   STATUS[506].TimeStamp := 16#0000;
   STATUS[507].VALUE := 0.0;
   STATUS[507].TRIGVALUE := 0.0;
   STATUS[507].EXT.AlarmWarnUnAck := FALSE;
   STATUS[507].EXT.AckRequired := FALSE;
   STATUS[507].EXT.Maintanence := FALSE;
   STATUS[507].EXT.Operation := FALSE;
   STATUS[507].EXT.Forced := FALSE;
   STATUS[507].EXT.BIT29 := FALSE;
   STATUS[507].EXT.BIT30 := FALSE;
   STATUS[507].EXT.BIT31 := FALSE;
   STATUS[507].EXT.ModeBit1 := FALSE;
   STATUS[507].EXT.ModeBit2 := FALSE;
   STATUS[507].EXT.ModeBit3 := FALSE;
   STATUS[507].EXT.BIT19 := FALSE;
   STATUS[507].EXT.BIT20 := FALSE;
   STATUS[507].EXT.AlarmSuppressed := FALSE;
   STATUS[507].EXT.AlarmPrsent := FALSE;
   STATUS[507].EXT.AlarmFailUnAck := FALSE;
   STATUS[507].Status := 0;
   STATUS[507].TimeStamp := 16#0000;
   STATUS[508].VALUE := 0.0;
   STATUS[508].TRIGVALUE := 0.0;
   STATUS[508].EXT.AlarmWarnUnAck := FALSE;
   STATUS[508].EXT.AckRequired := FALSE;
   STATUS[508].EXT.Maintanence := FALSE;
   STATUS[508].EXT.Operation := FALSE;
   STATUS[508].EXT.Forced := FALSE;
   STATUS[508].EXT.BIT29 := FALSE;
   STATUS[508].EXT.BIT30 := FALSE;
   STATUS[508].EXT.BIT31 := FALSE;
   STATUS[508].EXT.ModeBit1 := FALSE;
   STATUS[508].EXT.ModeBit2 := FALSE;
   STATUS[508].EXT.ModeBit3 := FALSE;
   STATUS[508].EXT.BIT19 := FALSE;
   STATUS[508].EXT.BIT20 := FALSE;
   STATUS[508].EXT.AlarmSuppressed := FALSE;
   STATUS[508].EXT.AlarmPrsent := FALSE;
   STATUS[508].EXT.AlarmFailUnAck := FALSE;
   STATUS[508].Status := 0;
   STATUS[508].TimeStamp := 16#0000;
   STATUS[509].VALUE := 0.0;
   STATUS[509].TRIGVALUE := 0.0;
   STATUS[509].EXT.AlarmWarnUnAck := FALSE;
   STATUS[509].EXT.AckRequired := FALSE;
   STATUS[509].EXT.Maintanence := FALSE;
   STATUS[509].EXT.Operation := FALSE;
   STATUS[509].EXT.Forced := FALSE;
   STATUS[509].EXT.BIT29 := FALSE;
   STATUS[509].EXT.BIT30 := FALSE;
   STATUS[509].EXT.BIT31 := FALSE;
   STATUS[509].EXT.ModeBit1 := FALSE;
   STATUS[509].EXT.ModeBit2 := FALSE;
   STATUS[509].EXT.ModeBit3 := FALSE;
   STATUS[509].EXT.BIT19 := FALSE;
   STATUS[509].EXT.BIT20 := FALSE;
   STATUS[509].EXT.AlarmSuppressed := FALSE;
   STATUS[509].EXT.AlarmPrsent := FALSE;
   STATUS[509].EXT.AlarmFailUnAck := FALSE;
   STATUS[509].Status := 0;
   STATUS[509].TimeStamp := 16#0000;
   STATUS[510].VALUE := 0.0;
   STATUS[510].TRIGVALUE := 0.0;
   STATUS[510].EXT.AlarmWarnUnAck := FALSE;
   STATUS[510].EXT.AckRequired := FALSE;
   STATUS[510].EXT.Maintanence := FALSE;
   STATUS[510].EXT.Operation := FALSE;
   STATUS[510].EXT.Forced := FALSE;
   STATUS[510].EXT.BIT29 := FALSE;
   STATUS[510].EXT.BIT30 := FALSE;
   STATUS[510].EXT.BIT31 := FALSE;
   STATUS[510].EXT.ModeBit1 := FALSE;
   STATUS[510].EXT.ModeBit2 := FALSE;
   STATUS[510].EXT.ModeBit3 := FALSE;
   STATUS[510].EXT.BIT19 := FALSE;
   STATUS[510].EXT.BIT20 := FALSE;
   STATUS[510].EXT.AlarmSuppressed := FALSE;
   STATUS[510].EXT.AlarmPrsent := FALSE;
   STATUS[510].EXT.AlarmFailUnAck := FALSE;
   STATUS[510].Status := 0;
   STATUS[510].TimeStamp := 16#0000;
   STATUS[511].VALUE := 0.0;
   STATUS[511].TRIGVALUE := 0.0;
   STATUS[511].EXT.AlarmWarnUnAck := FALSE;
   STATUS[511].EXT.AckRequired := FALSE;
   STATUS[511].EXT.Maintanence := FALSE;
   STATUS[511].EXT.Operation := FALSE;
   STATUS[511].EXT.Forced := FALSE;
   STATUS[511].EXT.BIT29 := FALSE;
   STATUS[511].EXT.BIT30 := FALSE;
   STATUS[511].EXT.BIT31 := FALSE;
   STATUS[511].EXT.ModeBit1 := FALSE;
   STATUS[511].EXT.ModeBit2 := FALSE;
   STATUS[511].EXT.ModeBit3 := FALSE;
   STATUS[511].EXT.BIT19 := FALSE;
   STATUS[511].EXT.BIT20 := FALSE;
   STATUS[511].EXT.AlarmSuppressed := FALSE;
   STATUS[511].EXT.AlarmPrsent := FALSE;
   STATUS[511].EXT.AlarmFailUnAck := FALSE;
   STATUS[511].Status := 0;
   STATUS[511].TimeStamp := 16#0000;
   STATUS[512].VALUE := 0.0;
   STATUS[512].TRIGVALUE := 0.0;
   STATUS[512].EXT.AlarmWarnUnAck := FALSE;
   STATUS[512].EXT.AckRequired := FALSE;
   STATUS[512].EXT.Maintanence := FALSE;
   STATUS[512].EXT.Operation := FALSE;
   STATUS[512].EXT.Forced := FALSE;
   STATUS[512].EXT.BIT29 := FALSE;
   STATUS[512].EXT.BIT30 := FALSE;
   STATUS[512].EXT.BIT31 := FALSE;
   STATUS[512].EXT.ModeBit1 := FALSE;
   STATUS[512].EXT.ModeBit2 := FALSE;
   STATUS[512].EXT.ModeBit3 := FALSE;
   STATUS[512].EXT.BIT19 := FALSE;
   STATUS[512].EXT.BIT20 := FALSE;
   STATUS[512].EXT.AlarmSuppressed := FALSE;
   STATUS[512].EXT.AlarmPrsent := FALSE;
   STATUS[512].EXT.AlarmFailUnAck := FALSE;
   STATUS[512].Status := 0;
   STATUS[512].TimeStamp := 16#0000;
   STATUS[513].VALUE := 0.0;
   STATUS[513].TRIGVALUE := 0.0;
   STATUS[513].EXT.AlarmWarnUnAck := FALSE;
   STATUS[513].EXT.AckRequired := FALSE;
   STATUS[513].EXT.Maintanence := FALSE;
   STATUS[513].EXT.Operation := FALSE;
   STATUS[513].EXT.Forced := FALSE;
   STATUS[513].EXT.BIT29 := FALSE;
   STATUS[513].EXT.BIT30 := FALSE;
   STATUS[513].EXT.BIT31 := FALSE;
   STATUS[513].EXT.ModeBit1 := FALSE;
   STATUS[513].EXT.ModeBit2 := FALSE;
   STATUS[513].EXT.ModeBit3 := FALSE;
   STATUS[513].EXT.BIT19 := FALSE;
   STATUS[513].EXT.BIT20 := FALSE;
   STATUS[513].EXT.AlarmSuppressed := FALSE;
   STATUS[513].EXT.AlarmPrsent := FALSE;
   STATUS[513].EXT.AlarmFailUnAck := FALSE;
   STATUS[513].Status := 0;
   STATUS[513].TimeStamp := 16#0000;
   STATUS[514].VALUE := 0.0;
   STATUS[514].TRIGVALUE := 0.0;
   STATUS[514].EXT.AlarmWarnUnAck := FALSE;
   STATUS[514].EXT.AckRequired := FALSE;
   STATUS[514].EXT.Maintanence := FALSE;
   STATUS[514].EXT.Operation := FALSE;
   STATUS[514].EXT.Forced := FALSE;
   STATUS[514].EXT.BIT29 := FALSE;
   STATUS[514].EXT.BIT30 := FALSE;
   STATUS[514].EXT.BIT31 := FALSE;
   STATUS[514].EXT.ModeBit1 := FALSE;
   STATUS[514].EXT.ModeBit2 := FALSE;
   STATUS[514].EXT.ModeBit3 := FALSE;
   STATUS[514].EXT.BIT19 := FALSE;
   STATUS[514].EXT.BIT20 := FALSE;
   STATUS[514].EXT.AlarmSuppressed := FALSE;
   STATUS[514].EXT.AlarmPrsent := FALSE;
   STATUS[514].EXT.AlarmFailUnAck := FALSE;
   STATUS[514].Status := 0;
   STATUS[514].TimeStamp := 16#0000;
   STATUS[515].VALUE := 0.0;
   STATUS[515].TRIGVALUE := 0.0;
   STATUS[515].EXT.AlarmWarnUnAck := FALSE;
   STATUS[515].EXT.AckRequired := FALSE;
   STATUS[515].EXT.Maintanence := FALSE;
   STATUS[515].EXT.Operation := FALSE;
   STATUS[515].EXT.Forced := FALSE;
   STATUS[515].EXT.BIT29 := FALSE;
   STATUS[515].EXT.BIT30 := FALSE;
   STATUS[515].EXT.BIT31 := FALSE;
   STATUS[515].EXT.ModeBit1 := FALSE;
   STATUS[515].EXT.ModeBit2 := FALSE;
   STATUS[515].EXT.ModeBit3 := FALSE;
   STATUS[515].EXT.BIT19 := FALSE;
   STATUS[515].EXT.BIT20 := FALSE;
   STATUS[515].EXT.AlarmSuppressed := FALSE;
   STATUS[515].EXT.AlarmPrsent := FALSE;
   STATUS[515].EXT.AlarmFailUnAck := FALSE;
   STATUS[515].Status := 0;
   STATUS[515].TimeStamp := 16#0000;
   STATUS[516].VALUE := 0.0;
   STATUS[516].TRIGVALUE := 0.0;
   STATUS[516].EXT.AlarmWarnUnAck := FALSE;
   STATUS[516].EXT.AckRequired := FALSE;
   STATUS[516].EXT.Maintanence := FALSE;
   STATUS[516].EXT.Operation := FALSE;
   STATUS[516].EXT.Forced := FALSE;
   STATUS[516].EXT.BIT29 := FALSE;
   STATUS[516].EXT.BIT30 := FALSE;
   STATUS[516].EXT.BIT31 := FALSE;
   STATUS[516].EXT.ModeBit1 := FALSE;
   STATUS[516].EXT.ModeBit2 := FALSE;
   STATUS[516].EXT.ModeBit3 := FALSE;
   STATUS[516].EXT.BIT19 := FALSE;
   STATUS[516].EXT.BIT20 := FALSE;
   STATUS[516].EXT.AlarmSuppressed := FALSE;
   STATUS[516].EXT.AlarmPrsent := FALSE;
   STATUS[516].EXT.AlarmFailUnAck := FALSE;
   STATUS[516].Status := 0;
   STATUS[516].TimeStamp := 16#0000;
   STATUS[517].VALUE := 0.0;
   STATUS[517].TRIGVALUE := 0.0;
   STATUS[517].EXT.AlarmWarnUnAck := FALSE;
   STATUS[517].EXT.AckRequired := FALSE;
   STATUS[517].EXT.Maintanence := FALSE;
   STATUS[517].EXT.Operation := FALSE;
   STATUS[517].EXT.Forced := FALSE;
   STATUS[517].EXT.BIT29 := FALSE;
   STATUS[517].EXT.BIT30 := FALSE;
   STATUS[517].EXT.BIT31 := FALSE;
   STATUS[517].EXT.ModeBit1 := FALSE;
   STATUS[517].EXT.ModeBit2 := FALSE;
   STATUS[517].EXT.ModeBit3 := FALSE;
   STATUS[517].EXT.BIT19 := FALSE;
   STATUS[517].EXT.BIT20 := FALSE;
   STATUS[517].EXT.AlarmSuppressed := FALSE;
   STATUS[517].EXT.AlarmPrsent := FALSE;
   STATUS[517].EXT.AlarmFailUnAck := FALSE;
   STATUS[517].Status := 0;
   STATUS[517].TimeStamp := 16#0000;
   STATUS[518].VALUE := 0.0;
   STATUS[518].TRIGVALUE := 0.0;
   STATUS[518].EXT.AlarmWarnUnAck := FALSE;
   STATUS[518].EXT.AckRequired := FALSE;
   STATUS[518].EXT.Maintanence := FALSE;
   STATUS[518].EXT.Operation := FALSE;
   STATUS[518].EXT.Forced := FALSE;
   STATUS[518].EXT.BIT29 := FALSE;
   STATUS[518].EXT.BIT30 := FALSE;
   STATUS[518].EXT.BIT31 := FALSE;
   STATUS[518].EXT.ModeBit1 := FALSE;
   STATUS[518].EXT.ModeBit2 := FALSE;
   STATUS[518].EXT.ModeBit3 := FALSE;
   STATUS[518].EXT.BIT19 := FALSE;
   STATUS[518].EXT.BIT20 := FALSE;
   STATUS[518].EXT.AlarmSuppressed := FALSE;
   STATUS[518].EXT.AlarmPrsent := FALSE;
   STATUS[518].EXT.AlarmFailUnAck := FALSE;
   STATUS[518].Status := 0;
   STATUS[518].TimeStamp := 16#0000;
   STATUS[519].VALUE := 0.0;
   STATUS[519].TRIGVALUE := 0.0;
   STATUS[519].EXT.AlarmWarnUnAck := FALSE;
   STATUS[519].EXT.AckRequired := FALSE;
   STATUS[519].EXT.Maintanence := FALSE;
   STATUS[519].EXT.Operation := FALSE;
   STATUS[519].EXT.Forced := FALSE;
   STATUS[519].EXT.BIT29 := FALSE;
   STATUS[519].EXT.BIT30 := FALSE;
   STATUS[519].EXT.BIT31 := FALSE;
   STATUS[519].EXT.ModeBit1 := FALSE;
   STATUS[519].EXT.ModeBit2 := FALSE;
   STATUS[519].EXT.ModeBit3 := FALSE;
   STATUS[519].EXT.BIT19 := FALSE;
   STATUS[519].EXT.BIT20 := FALSE;
   STATUS[519].EXT.AlarmSuppressed := FALSE;
   STATUS[519].EXT.AlarmPrsent := FALSE;
   STATUS[519].EXT.AlarmFailUnAck := FALSE;
   STATUS[519].Status := 0;
   STATUS[519].TimeStamp := 16#0000;
   STATUS[520].VALUE := 0.0;
   STATUS[520].TRIGVALUE := 0.0;
   STATUS[520].EXT.AlarmWarnUnAck := FALSE;
   STATUS[520].EXT.AckRequired := FALSE;
   STATUS[520].EXT.Maintanence := FALSE;
   STATUS[520].EXT.Operation := FALSE;
   STATUS[520].EXT.Forced := FALSE;
   STATUS[520].EXT.BIT29 := FALSE;
   STATUS[520].EXT.BIT30 := FALSE;
   STATUS[520].EXT.BIT31 := FALSE;
   STATUS[520].EXT.ModeBit1 := FALSE;
   STATUS[520].EXT.ModeBit2 := FALSE;
   STATUS[520].EXT.ModeBit3 := FALSE;
   STATUS[520].EXT.BIT19 := FALSE;
   STATUS[520].EXT.BIT20 := FALSE;
   STATUS[520].EXT.AlarmSuppressed := FALSE;
   STATUS[520].EXT.AlarmPrsent := FALSE;
   STATUS[520].EXT.AlarmFailUnAck := FALSE;
   STATUS[520].Status := 0;
   STATUS[520].TimeStamp := 16#0000;
   STATUS[521].VALUE := 0.0;
   STATUS[521].TRIGVALUE := 0.0;
   STATUS[521].EXT.AlarmWarnUnAck := FALSE;
   STATUS[521].EXT.AckRequired := FALSE;
   STATUS[521].EXT.Maintanence := FALSE;
   STATUS[521].EXT.Operation := FALSE;
   STATUS[521].EXT.Forced := FALSE;
   STATUS[521].EXT.BIT29 := FALSE;
   STATUS[521].EXT.BIT30 := FALSE;
   STATUS[521].EXT.BIT31 := FALSE;
   STATUS[521].EXT.ModeBit1 := FALSE;
   STATUS[521].EXT.ModeBit2 := FALSE;
   STATUS[521].EXT.ModeBit3 := FALSE;
   STATUS[521].EXT.BIT19 := FALSE;
   STATUS[521].EXT.BIT20 := FALSE;
   STATUS[521].EXT.AlarmSuppressed := FALSE;
   STATUS[521].EXT.AlarmPrsent := FALSE;
   STATUS[521].EXT.AlarmFailUnAck := FALSE;
   STATUS[521].Status := 0;
   STATUS[521].TimeStamp := 16#0000;
   STATUS[522].VALUE := 0.0;
   STATUS[522].TRIGVALUE := 0.0;
   STATUS[522].EXT.AlarmWarnUnAck := FALSE;
   STATUS[522].EXT.AckRequired := FALSE;
   STATUS[522].EXT.Maintanence := FALSE;
   STATUS[522].EXT.Operation := FALSE;
   STATUS[522].EXT.Forced := FALSE;
   STATUS[522].EXT.BIT29 := FALSE;
   STATUS[522].EXT.BIT30 := FALSE;
   STATUS[522].EXT.BIT31 := FALSE;
   STATUS[522].EXT.ModeBit1 := FALSE;
   STATUS[522].EXT.ModeBit2 := FALSE;
   STATUS[522].EXT.ModeBit3 := FALSE;
   STATUS[522].EXT.BIT19 := FALSE;
   STATUS[522].EXT.BIT20 := FALSE;
   STATUS[522].EXT.AlarmSuppressed := FALSE;
   STATUS[522].EXT.AlarmPrsent := FALSE;
   STATUS[522].EXT.AlarmFailUnAck := FALSE;
   STATUS[522].Status := 0;
   STATUS[522].TimeStamp := 16#0000;
   STATUS[523].VALUE := 0.0;
   STATUS[523].TRIGVALUE := 0.0;
   STATUS[523].EXT.AlarmWarnUnAck := FALSE;
   STATUS[523].EXT.AckRequired := FALSE;
   STATUS[523].EXT.Maintanence := FALSE;
   STATUS[523].EXT.Operation := FALSE;
   STATUS[523].EXT.Forced := FALSE;
   STATUS[523].EXT.BIT29 := FALSE;
   STATUS[523].EXT.BIT30 := FALSE;
   STATUS[523].EXT.BIT31 := FALSE;
   STATUS[523].EXT.ModeBit1 := FALSE;
   STATUS[523].EXT.ModeBit2 := FALSE;
   STATUS[523].EXT.ModeBit3 := FALSE;
   STATUS[523].EXT.BIT19 := FALSE;
   STATUS[523].EXT.BIT20 := FALSE;
   STATUS[523].EXT.AlarmSuppressed := FALSE;
   STATUS[523].EXT.AlarmPrsent := FALSE;
   STATUS[523].EXT.AlarmFailUnAck := FALSE;
   STATUS[523].Status := 0;
   STATUS[523].TimeStamp := 16#0000;
   STATUS[524].VALUE := 0.0;
   STATUS[524].TRIGVALUE := 0.0;
   STATUS[524].EXT.AlarmWarnUnAck := FALSE;
   STATUS[524].EXT.AckRequired := FALSE;
   STATUS[524].EXT.Maintanence := FALSE;
   STATUS[524].EXT.Operation := FALSE;
   STATUS[524].EXT.Forced := FALSE;
   STATUS[524].EXT.BIT29 := FALSE;
   STATUS[524].EXT.BIT30 := FALSE;
   STATUS[524].EXT.BIT31 := FALSE;
   STATUS[524].EXT.ModeBit1 := FALSE;
   STATUS[524].EXT.ModeBit2 := FALSE;
   STATUS[524].EXT.ModeBit3 := FALSE;
   STATUS[524].EXT.BIT19 := FALSE;
   STATUS[524].EXT.BIT20 := FALSE;
   STATUS[524].EXT.AlarmSuppressed := FALSE;
   STATUS[524].EXT.AlarmPrsent := FALSE;
   STATUS[524].EXT.AlarmFailUnAck := FALSE;
   STATUS[524].Status := 0;
   STATUS[524].TimeStamp := 16#0000;
   STATUS[525].VALUE := 0.0;
   STATUS[525].TRIGVALUE := 0.0;
   STATUS[525].EXT.AlarmWarnUnAck := FALSE;
   STATUS[525].EXT.AckRequired := FALSE;
   STATUS[525].EXT.Maintanence := FALSE;
   STATUS[525].EXT.Operation := FALSE;
   STATUS[525].EXT.Forced := FALSE;
   STATUS[525].EXT.BIT29 := FALSE;
   STATUS[525].EXT.BIT30 := FALSE;
   STATUS[525].EXT.BIT31 := FALSE;
   STATUS[525].EXT.ModeBit1 := FALSE;
   STATUS[525].EXT.ModeBit2 := FALSE;
   STATUS[525].EXT.ModeBit3 := FALSE;
   STATUS[525].EXT.BIT19 := FALSE;
   STATUS[525].EXT.BIT20 := FALSE;
   STATUS[525].EXT.AlarmSuppressed := FALSE;
   STATUS[525].EXT.AlarmPrsent := FALSE;
   STATUS[525].EXT.AlarmFailUnAck := FALSE;
   STATUS[525].Status := 0;
   STATUS[525].TimeStamp := 16#0000;
   STATUS[526].VALUE := 0.0;
   STATUS[526].TRIGVALUE := 0.0;
   STATUS[526].EXT.AlarmWarnUnAck := FALSE;
   STATUS[526].EXT.AckRequired := FALSE;
   STATUS[526].EXT.Maintanence := FALSE;
   STATUS[526].EXT.Operation := FALSE;
   STATUS[526].EXT.Forced := FALSE;
   STATUS[526].EXT.BIT29 := FALSE;
   STATUS[526].EXT.BIT30 := FALSE;
   STATUS[526].EXT.BIT31 := FALSE;
   STATUS[526].EXT.ModeBit1 := FALSE;
   STATUS[526].EXT.ModeBit2 := FALSE;
   STATUS[526].EXT.ModeBit3 := FALSE;
   STATUS[526].EXT.BIT19 := FALSE;
   STATUS[526].EXT.BIT20 := FALSE;
   STATUS[526].EXT.AlarmSuppressed := FALSE;
   STATUS[526].EXT.AlarmPrsent := FALSE;
   STATUS[526].EXT.AlarmFailUnAck := FALSE;
   STATUS[526].Status := 0;
   STATUS[526].TimeStamp := 16#0000;
   STATUS[527].VALUE := 0.0;
   STATUS[527].TRIGVALUE := 0.0;
   STATUS[527].EXT.AlarmWarnUnAck := FALSE;
   STATUS[527].EXT.AckRequired := FALSE;
   STATUS[527].EXT.Maintanence := FALSE;
   STATUS[527].EXT.Operation := FALSE;
   STATUS[527].EXT.Forced := FALSE;
   STATUS[527].EXT.BIT29 := FALSE;
   STATUS[527].EXT.BIT30 := FALSE;
   STATUS[527].EXT.BIT31 := FALSE;
   STATUS[527].EXT.ModeBit1 := FALSE;
   STATUS[527].EXT.ModeBit2 := FALSE;
   STATUS[527].EXT.ModeBit3 := FALSE;
   STATUS[527].EXT.BIT19 := FALSE;
   STATUS[527].EXT.BIT20 := FALSE;
   STATUS[527].EXT.AlarmSuppressed := FALSE;
   STATUS[527].EXT.AlarmPrsent := FALSE;
   STATUS[527].EXT.AlarmFailUnAck := FALSE;
   STATUS[527].Status := 0;
   STATUS[527].TimeStamp := 16#0000;
   STATUS[528].VALUE := 0.0;
   STATUS[528].TRIGVALUE := 0.0;
   STATUS[528].EXT.AlarmWarnUnAck := FALSE;
   STATUS[528].EXT.AckRequired := FALSE;
   STATUS[528].EXT.Maintanence := FALSE;
   STATUS[528].EXT.Operation := FALSE;
   STATUS[528].EXT.Forced := FALSE;
   STATUS[528].EXT.BIT29 := FALSE;
   STATUS[528].EXT.BIT30 := FALSE;
   STATUS[528].EXT.BIT31 := FALSE;
   STATUS[528].EXT.ModeBit1 := FALSE;
   STATUS[528].EXT.ModeBit2 := FALSE;
   STATUS[528].EXT.ModeBit3 := FALSE;
   STATUS[528].EXT.BIT19 := FALSE;
   STATUS[528].EXT.BIT20 := FALSE;
   STATUS[528].EXT.AlarmSuppressed := FALSE;
   STATUS[528].EXT.AlarmPrsent := FALSE;
   STATUS[528].EXT.AlarmFailUnAck := FALSE;
   STATUS[528].Status := 0;
   STATUS[528].TimeStamp := 16#0000;
   STATUS[529].VALUE := 0.0;
   STATUS[529].TRIGVALUE := 0.0;
   STATUS[529].EXT.AlarmWarnUnAck := FALSE;
   STATUS[529].EXT.AckRequired := FALSE;
   STATUS[529].EXT.Maintanence := FALSE;
   STATUS[529].EXT.Operation := FALSE;
   STATUS[529].EXT.Forced := FALSE;
   STATUS[529].EXT.BIT29 := FALSE;
   STATUS[529].EXT.BIT30 := FALSE;
   STATUS[529].EXT.BIT31 := FALSE;
   STATUS[529].EXT.ModeBit1 := FALSE;
   STATUS[529].EXT.ModeBit2 := FALSE;
   STATUS[529].EXT.ModeBit3 := FALSE;
   STATUS[529].EXT.BIT19 := FALSE;
   STATUS[529].EXT.BIT20 := FALSE;
   STATUS[529].EXT.AlarmSuppressed := FALSE;
   STATUS[529].EXT.AlarmPrsent := FALSE;
   STATUS[529].EXT.AlarmFailUnAck := FALSE;
   STATUS[529].Status := 0;
   STATUS[529].TimeStamp := 16#0000;
   STATUS[530].VALUE := 0.0;
   STATUS[530].TRIGVALUE := 0.0;
   STATUS[530].EXT.AlarmWarnUnAck := FALSE;
   STATUS[530].EXT.AckRequired := FALSE;
   STATUS[530].EXT.Maintanence := FALSE;
   STATUS[530].EXT.Operation := FALSE;
   STATUS[530].EXT.Forced := FALSE;
   STATUS[530].EXT.BIT29 := FALSE;
   STATUS[530].EXT.BIT30 := FALSE;
   STATUS[530].EXT.BIT31 := FALSE;
   STATUS[530].EXT.ModeBit1 := FALSE;
   STATUS[530].EXT.ModeBit2 := FALSE;
   STATUS[530].EXT.ModeBit3 := FALSE;
   STATUS[530].EXT.BIT19 := FALSE;
   STATUS[530].EXT.BIT20 := FALSE;
   STATUS[530].EXT.AlarmSuppressed := FALSE;
   STATUS[530].EXT.AlarmPrsent := FALSE;
   STATUS[530].EXT.AlarmFailUnAck := FALSE;
   STATUS[530].Status := 0;
   STATUS[530].TimeStamp := 16#0000;
   STATUS[531].VALUE := 0.0;
   STATUS[531].TRIGVALUE := 0.0;
   STATUS[531].EXT.AlarmWarnUnAck := FALSE;
   STATUS[531].EXT.AckRequired := FALSE;
   STATUS[531].EXT.Maintanence := FALSE;
   STATUS[531].EXT.Operation := FALSE;
   STATUS[531].EXT.Forced := FALSE;
   STATUS[531].EXT.BIT29 := FALSE;
   STATUS[531].EXT.BIT30 := FALSE;
   STATUS[531].EXT.BIT31 := FALSE;
   STATUS[531].EXT.ModeBit1 := FALSE;
   STATUS[531].EXT.ModeBit2 := FALSE;
   STATUS[531].EXT.ModeBit3 := FALSE;
   STATUS[531].EXT.BIT19 := FALSE;
   STATUS[531].EXT.BIT20 := FALSE;
   STATUS[531].EXT.AlarmSuppressed := FALSE;
   STATUS[531].EXT.AlarmPrsent := FALSE;
   STATUS[531].EXT.AlarmFailUnAck := FALSE;
   STATUS[531].Status := 0;
   STATUS[531].TimeStamp := 16#0000;
   STATUS[532].VALUE := 0.0;
   STATUS[532].TRIGVALUE := 0.0;
   STATUS[532].EXT.AlarmWarnUnAck := FALSE;
   STATUS[532].EXT.AckRequired := FALSE;
   STATUS[532].EXT.Maintanence := FALSE;
   STATUS[532].EXT.Operation := FALSE;
   STATUS[532].EXT.Forced := FALSE;
   STATUS[532].EXT.BIT29 := FALSE;
   STATUS[532].EXT.BIT30 := FALSE;
   STATUS[532].EXT.BIT31 := FALSE;
   STATUS[532].EXT.ModeBit1 := FALSE;
   STATUS[532].EXT.ModeBit2 := FALSE;
   STATUS[532].EXT.ModeBit3 := FALSE;
   STATUS[532].EXT.BIT19 := FALSE;
   STATUS[532].EXT.BIT20 := FALSE;
   STATUS[532].EXT.AlarmSuppressed := FALSE;
   STATUS[532].EXT.AlarmPrsent := FALSE;
   STATUS[532].EXT.AlarmFailUnAck := FALSE;
   STATUS[532].Status := 0;
   STATUS[532].TimeStamp := 16#0000;
   STATUS[533].VALUE := 0.0;
   STATUS[533].TRIGVALUE := 0.0;
   STATUS[533].EXT.AlarmWarnUnAck := FALSE;
   STATUS[533].EXT.AckRequired := FALSE;
   STATUS[533].EXT.Maintanence := FALSE;
   STATUS[533].EXT.Operation := FALSE;
   STATUS[533].EXT.Forced := FALSE;
   STATUS[533].EXT.BIT29 := FALSE;
   STATUS[533].EXT.BIT30 := FALSE;
   STATUS[533].EXT.BIT31 := FALSE;
   STATUS[533].EXT.ModeBit1 := FALSE;
   STATUS[533].EXT.ModeBit2 := FALSE;
   STATUS[533].EXT.ModeBit3 := FALSE;
   STATUS[533].EXT.BIT19 := FALSE;
   STATUS[533].EXT.BIT20 := FALSE;
   STATUS[533].EXT.AlarmSuppressed := FALSE;
   STATUS[533].EXT.AlarmPrsent := FALSE;
   STATUS[533].EXT.AlarmFailUnAck := FALSE;
   STATUS[533].Status := 0;
   STATUS[533].TimeStamp := 16#0000;
   STATUS[534].VALUE := 0.0;
   STATUS[534].TRIGVALUE := 0.0;
   STATUS[534].EXT.AlarmWarnUnAck := FALSE;
   STATUS[534].EXT.AckRequired := FALSE;
   STATUS[534].EXT.Maintanence := FALSE;
   STATUS[534].EXT.Operation := FALSE;
   STATUS[534].EXT.Forced := FALSE;
   STATUS[534].EXT.BIT29 := FALSE;
   STATUS[534].EXT.BIT30 := FALSE;
   STATUS[534].EXT.BIT31 := FALSE;
   STATUS[534].EXT.ModeBit1 := FALSE;
   STATUS[534].EXT.ModeBit2 := FALSE;
   STATUS[534].EXT.ModeBit3 := FALSE;
   STATUS[534].EXT.BIT19 := FALSE;
   STATUS[534].EXT.BIT20 := FALSE;
   STATUS[534].EXT.AlarmSuppressed := FALSE;
   STATUS[534].EXT.AlarmPrsent := FALSE;
   STATUS[534].EXT.AlarmFailUnAck := FALSE;
   STATUS[534].Status := 0;
   STATUS[534].TimeStamp := 16#0000;
   STATUS[535].VALUE := 0.0;
   STATUS[535].TRIGVALUE := 0.0;
   STATUS[535].EXT.AlarmWarnUnAck := FALSE;
   STATUS[535].EXT.AckRequired := FALSE;
   STATUS[535].EXT.Maintanence := FALSE;
   STATUS[535].EXT.Operation := FALSE;
   STATUS[535].EXT.Forced := FALSE;
   STATUS[535].EXT.BIT29 := FALSE;
   STATUS[535].EXT.BIT30 := FALSE;
   STATUS[535].EXT.BIT31 := FALSE;
   STATUS[535].EXT.ModeBit1 := FALSE;
   STATUS[535].EXT.ModeBit2 := FALSE;
   STATUS[535].EXT.ModeBit3 := FALSE;
   STATUS[535].EXT.BIT19 := FALSE;
   STATUS[535].EXT.BIT20 := FALSE;
   STATUS[535].EXT.AlarmSuppressed := FALSE;
   STATUS[535].EXT.AlarmPrsent := FALSE;
   STATUS[535].EXT.AlarmFailUnAck := FALSE;
   STATUS[535].Status := 0;
   STATUS[535].TimeStamp := 16#0000;
   STATUS[536].VALUE := 0.0;
   STATUS[536].TRIGVALUE := 0.0;
   STATUS[536].EXT.AlarmWarnUnAck := FALSE;
   STATUS[536].EXT.AckRequired := FALSE;
   STATUS[536].EXT.Maintanence := FALSE;
   STATUS[536].EXT.Operation := FALSE;
   STATUS[536].EXT.Forced := FALSE;
   STATUS[536].EXT.BIT29 := FALSE;
   STATUS[536].EXT.BIT30 := FALSE;
   STATUS[536].EXT.BIT31 := FALSE;
   STATUS[536].EXT.ModeBit1 := FALSE;
   STATUS[536].EXT.ModeBit2 := FALSE;
   STATUS[536].EXT.ModeBit3 := FALSE;
   STATUS[536].EXT.BIT19 := FALSE;
   STATUS[536].EXT.BIT20 := FALSE;
   STATUS[536].EXT.AlarmSuppressed := FALSE;
   STATUS[536].EXT.AlarmPrsent := FALSE;
   STATUS[536].EXT.AlarmFailUnAck := FALSE;
   STATUS[536].Status := 0;
   STATUS[536].TimeStamp := 16#0000;
   STATUS[537].VALUE := 0.0;
   STATUS[537].TRIGVALUE := 0.0;
   STATUS[537].EXT.AlarmWarnUnAck := FALSE;
   STATUS[537].EXT.AckRequired := FALSE;
   STATUS[537].EXT.Maintanence := FALSE;
   STATUS[537].EXT.Operation := FALSE;
   STATUS[537].EXT.Forced := FALSE;
   STATUS[537].EXT.BIT29 := FALSE;
   STATUS[537].EXT.BIT30 := FALSE;
   STATUS[537].EXT.BIT31 := FALSE;
   STATUS[537].EXT.ModeBit1 := FALSE;
   STATUS[537].EXT.ModeBit2 := FALSE;
   STATUS[537].EXT.ModeBit3 := FALSE;
   STATUS[537].EXT.BIT19 := FALSE;
   STATUS[537].EXT.BIT20 := FALSE;
   STATUS[537].EXT.AlarmSuppressed := FALSE;
   STATUS[537].EXT.AlarmPrsent := FALSE;
   STATUS[537].EXT.AlarmFailUnAck := FALSE;
   STATUS[537].Status := 0;
   STATUS[537].TimeStamp := 16#0000;
   STATUS[538].VALUE := 0.0;
   STATUS[538].TRIGVALUE := 0.0;
   STATUS[538].EXT.AlarmWarnUnAck := FALSE;
   STATUS[538].EXT.AckRequired := FALSE;
   STATUS[538].EXT.Maintanence := FALSE;
   STATUS[538].EXT.Operation := FALSE;
   STATUS[538].EXT.Forced := FALSE;
   STATUS[538].EXT.BIT29 := FALSE;
   STATUS[538].EXT.BIT30 := FALSE;
   STATUS[538].EXT.BIT31 := FALSE;
   STATUS[538].EXT.ModeBit1 := FALSE;
   STATUS[538].EXT.ModeBit2 := FALSE;
   STATUS[538].EXT.ModeBit3 := FALSE;
   STATUS[538].EXT.BIT19 := FALSE;
   STATUS[538].EXT.BIT20 := FALSE;
   STATUS[538].EXT.AlarmSuppressed := FALSE;
   STATUS[538].EXT.AlarmPrsent := FALSE;
   STATUS[538].EXT.AlarmFailUnAck := FALSE;
   STATUS[538].Status := 0;
   STATUS[538].TimeStamp := 16#0000;
   STATUS[539].VALUE := 0.0;
   STATUS[539].TRIGVALUE := 0.0;
   STATUS[539].EXT.AlarmWarnUnAck := FALSE;
   STATUS[539].EXT.AckRequired := FALSE;
   STATUS[539].EXT.Maintanence := FALSE;
   STATUS[539].EXT.Operation := FALSE;
   STATUS[539].EXT.Forced := FALSE;
   STATUS[539].EXT.BIT29 := FALSE;
   STATUS[539].EXT.BIT30 := FALSE;
   STATUS[539].EXT.BIT31 := FALSE;
   STATUS[539].EXT.ModeBit1 := FALSE;
   STATUS[539].EXT.ModeBit2 := FALSE;
   STATUS[539].EXT.ModeBit3 := FALSE;
   STATUS[539].EXT.BIT19 := FALSE;
   STATUS[539].EXT.BIT20 := FALSE;
   STATUS[539].EXT.AlarmSuppressed := FALSE;
   STATUS[539].EXT.AlarmPrsent := FALSE;
   STATUS[539].EXT.AlarmFailUnAck := FALSE;
   STATUS[539].Status := 0;
   STATUS[539].TimeStamp := 16#0000;
   STATUS[540].VALUE := 0.0;
   STATUS[540].TRIGVALUE := 0.0;
   STATUS[540].EXT.AlarmWarnUnAck := FALSE;
   STATUS[540].EXT.AckRequired := FALSE;
   STATUS[540].EXT.Maintanence := FALSE;
   STATUS[540].EXT.Operation := FALSE;
   STATUS[540].EXT.Forced := FALSE;
   STATUS[540].EXT.BIT29 := FALSE;
   STATUS[540].EXT.BIT30 := FALSE;
   STATUS[540].EXT.BIT31 := FALSE;
   STATUS[540].EXT.ModeBit1 := FALSE;
   STATUS[540].EXT.ModeBit2 := FALSE;
   STATUS[540].EXT.ModeBit3 := FALSE;
   STATUS[540].EXT.BIT19 := FALSE;
   STATUS[540].EXT.BIT20 := FALSE;
   STATUS[540].EXT.AlarmSuppressed := FALSE;
   STATUS[540].EXT.AlarmPrsent := FALSE;
   STATUS[540].EXT.AlarmFailUnAck := FALSE;
   STATUS[540].Status := 0;
   STATUS[540].TimeStamp := 16#0000;
   STATUS[541].VALUE := 0.0;
   STATUS[541].TRIGVALUE := 0.0;
   STATUS[541].EXT.AlarmWarnUnAck := FALSE;
   STATUS[541].EXT.AckRequired := FALSE;
   STATUS[541].EXT.Maintanence := FALSE;
   STATUS[541].EXT.Operation := FALSE;
   STATUS[541].EXT.Forced := FALSE;
   STATUS[541].EXT.BIT29 := FALSE;
   STATUS[541].EXT.BIT30 := FALSE;
   STATUS[541].EXT.BIT31 := FALSE;
   STATUS[541].EXT.ModeBit1 := FALSE;
   STATUS[541].EXT.ModeBit2 := FALSE;
   STATUS[541].EXT.ModeBit3 := FALSE;
   STATUS[541].EXT.BIT19 := FALSE;
   STATUS[541].EXT.BIT20 := FALSE;
   STATUS[541].EXT.AlarmSuppressed := FALSE;
   STATUS[541].EXT.AlarmPrsent := FALSE;
   STATUS[541].EXT.AlarmFailUnAck := FALSE;
   STATUS[541].Status := 0;
   STATUS[541].TimeStamp := 16#0000;
   STATUS[542].VALUE := 0.0;
   STATUS[542].TRIGVALUE := 0.0;
   STATUS[542].EXT.AlarmWarnUnAck := FALSE;
   STATUS[542].EXT.AckRequired := FALSE;
   STATUS[542].EXT.Maintanence := FALSE;
   STATUS[542].EXT.Operation := FALSE;
   STATUS[542].EXT.Forced := FALSE;
   STATUS[542].EXT.BIT29 := FALSE;
   STATUS[542].EXT.BIT30 := FALSE;
   STATUS[542].EXT.BIT31 := FALSE;
   STATUS[542].EXT.ModeBit1 := FALSE;
   STATUS[542].EXT.ModeBit2 := FALSE;
   STATUS[542].EXT.ModeBit3 := FALSE;
   STATUS[542].EXT.BIT19 := FALSE;
   STATUS[542].EXT.BIT20 := FALSE;
   STATUS[542].EXT.AlarmSuppressed := FALSE;
   STATUS[542].EXT.AlarmPrsent := FALSE;
   STATUS[542].EXT.AlarmFailUnAck := FALSE;
   STATUS[542].Status := 0;
   STATUS[542].TimeStamp := 16#0000;
   STATUS[543].VALUE := 0.0;
   STATUS[543].TRIGVALUE := 0.0;
   STATUS[543].EXT.AlarmWarnUnAck := FALSE;
   STATUS[543].EXT.AckRequired := FALSE;
   STATUS[543].EXT.Maintanence := FALSE;
   STATUS[543].EXT.Operation := FALSE;
   STATUS[543].EXT.Forced := FALSE;
   STATUS[543].EXT.BIT29 := FALSE;
   STATUS[543].EXT.BIT30 := FALSE;
   STATUS[543].EXT.BIT31 := FALSE;
   STATUS[543].EXT.ModeBit1 := FALSE;
   STATUS[543].EXT.ModeBit2 := FALSE;
   STATUS[543].EXT.ModeBit3 := FALSE;
   STATUS[543].EXT.BIT19 := FALSE;
   STATUS[543].EXT.BIT20 := FALSE;
   STATUS[543].EXT.AlarmSuppressed := FALSE;
   STATUS[543].EXT.AlarmPrsent := FALSE;
   STATUS[543].EXT.AlarmFailUnAck := FALSE;
   STATUS[543].Status := 0;
   STATUS[543].TimeStamp := 16#0000;
   STATUS[544].VALUE := 0.0;
   STATUS[544].TRIGVALUE := 0.0;
   STATUS[544].EXT.AlarmWarnUnAck := FALSE;
   STATUS[544].EXT.AckRequired := FALSE;
   STATUS[544].EXT.Maintanence := FALSE;
   STATUS[544].EXT.Operation := FALSE;
   STATUS[544].EXT.Forced := FALSE;
   STATUS[544].EXT.BIT29 := FALSE;
   STATUS[544].EXT.BIT30 := FALSE;
   STATUS[544].EXT.BIT31 := FALSE;
   STATUS[544].EXT.ModeBit1 := FALSE;
   STATUS[544].EXT.ModeBit2 := FALSE;
   STATUS[544].EXT.ModeBit3 := FALSE;
   STATUS[544].EXT.BIT19 := FALSE;
   STATUS[544].EXT.BIT20 := FALSE;
   STATUS[544].EXT.AlarmSuppressed := FALSE;
   STATUS[544].EXT.AlarmPrsent := FALSE;
   STATUS[544].EXT.AlarmFailUnAck := FALSE;
   STATUS[544].Status := 0;
   STATUS[544].TimeStamp := 16#0000;
   STATUS[545].VALUE := 0.0;
   STATUS[545].TRIGVALUE := 0.0;
   STATUS[545].EXT.AlarmWarnUnAck := FALSE;
   STATUS[545].EXT.AckRequired := FALSE;
   STATUS[545].EXT.Maintanence := FALSE;
   STATUS[545].EXT.Operation := FALSE;
   STATUS[545].EXT.Forced := FALSE;
   STATUS[545].EXT.BIT29 := FALSE;
   STATUS[545].EXT.BIT30 := FALSE;
   STATUS[545].EXT.BIT31 := FALSE;
   STATUS[545].EXT.ModeBit1 := FALSE;
   STATUS[545].EXT.ModeBit2 := FALSE;
   STATUS[545].EXT.ModeBit3 := FALSE;
   STATUS[545].EXT.BIT19 := FALSE;
   STATUS[545].EXT.BIT20 := FALSE;
   STATUS[545].EXT.AlarmSuppressed := FALSE;
   STATUS[545].EXT.AlarmPrsent := FALSE;
   STATUS[545].EXT.AlarmFailUnAck := FALSE;
   STATUS[545].Status := 0;
   STATUS[545].TimeStamp := 16#0000;
   STATUS[546].VALUE := 0.0;
   STATUS[546].TRIGVALUE := 0.0;
   STATUS[546].EXT.AlarmWarnUnAck := FALSE;
   STATUS[546].EXT.AckRequired := FALSE;
   STATUS[546].EXT.Maintanence := FALSE;
   STATUS[546].EXT.Operation := FALSE;
   STATUS[546].EXT.Forced := FALSE;
   STATUS[546].EXT.BIT29 := FALSE;
   STATUS[546].EXT.BIT30 := FALSE;
   STATUS[546].EXT.BIT31 := FALSE;
   STATUS[546].EXT.ModeBit1 := FALSE;
   STATUS[546].EXT.ModeBit2 := FALSE;
   STATUS[546].EXT.ModeBit3 := FALSE;
   STATUS[546].EXT.BIT19 := FALSE;
   STATUS[546].EXT.BIT20 := FALSE;
   STATUS[546].EXT.AlarmSuppressed := FALSE;
   STATUS[546].EXT.AlarmPrsent := FALSE;
   STATUS[546].EXT.AlarmFailUnAck := FALSE;
   STATUS[546].Status := 0;
   STATUS[546].TimeStamp := 16#0000;
   STATUS[547].VALUE := 0.0;
   STATUS[547].TRIGVALUE := 0.0;
   STATUS[547].EXT.AlarmWarnUnAck := FALSE;
   STATUS[547].EXT.AckRequired := FALSE;
   STATUS[547].EXT.Maintanence := FALSE;
   STATUS[547].EXT.Operation := FALSE;
   STATUS[547].EXT.Forced := FALSE;
   STATUS[547].EXT.BIT29 := FALSE;
   STATUS[547].EXT.BIT30 := FALSE;
   STATUS[547].EXT.BIT31 := FALSE;
   STATUS[547].EXT.ModeBit1 := FALSE;
   STATUS[547].EXT.ModeBit2 := FALSE;
   STATUS[547].EXT.ModeBit3 := FALSE;
   STATUS[547].EXT.BIT19 := FALSE;
   STATUS[547].EXT.BIT20 := FALSE;
   STATUS[547].EXT.AlarmSuppressed := FALSE;
   STATUS[547].EXT.AlarmPrsent := FALSE;
   STATUS[547].EXT.AlarmFailUnAck := FALSE;
   STATUS[547].Status := 0;
   STATUS[547].TimeStamp := 16#0000;
   STATUS[548].VALUE := 0.0;
   STATUS[548].TRIGVALUE := 0.0;
   STATUS[548].EXT.AlarmWarnUnAck := FALSE;
   STATUS[548].EXT.AckRequired := FALSE;
   STATUS[548].EXT.Maintanence := FALSE;
   STATUS[548].EXT.Operation := FALSE;
   STATUS[548].EXT.Forced := FALSE;
   STATUS[548].EXT.BIT29 := FALSE;
   STATUS[548].EXT.BIT30 := FALSE;
   STATUS[548].EXT.BIT31 := FALSE;
   STATUS[548].EXT.ModeBit1 := FALSE;
   STATUS[548].EXT.ModeBit2 := FALSE;
   STATUS[548].EXT.ModeBit3 := FALSE;
   STATUS[548].EXT.BIT19 := FALSE;
   STATUS[548].EXT.BIT20 := FALSE;
   STATUS[548].EXT.AlarmSuppressed := FALSE;
   STATUS[548].EXT.AlarmPrsent := FALSE;
   STATUS[548].EXT.AlarmFailUnAck := FALSE;
   STATUS[548].Status := 0;
   STATUS[548].TimeStamp := 16#0000;
   STATUS[549].VALUE := 0.0;
   STATUS[549].TRIGVALUE := 0.0;
   STATUS[549].EXT.AlarmWarnUnAck := FALSE;
   STATUS[549].EXT.AckRequired := FALSE;
   STATUS[549].EXT.Maintanence := FALSE;
   STATUS[549].EXT.Operation := FALSE;
   STATUS[549].EXT.Forced := FALSE;
   STATUS[549].EXT.BIT29 := FALSE;
   STATUS[549].EXT.BIT30 := FALSE;
   STATUS[549].EXT.BIT31 := FALSE;
   STATUS[549].EXT.ModeBit1 := FALSE;
   STATUS[549].EXT.ModeBit2 := FALSE;
   STATUS[549].EXT.ModeBit3 := FALSE;
   STATUS[549].EXT.BIT19 := FALSE;
   STATUS[549].EXT.BIT20 := FALSE;
   STATUS[549].EXT.AlarmSuppressed := FALSE;
   STATUS[549].EXT.AlarmPrsent := FALSE;
   STATUS[549].EXT.AlarmFailUnAck := FALSE;
   STATUS[549].Status := 0;
   STATUS[549].TimeStamp := 16#0000;
   STATUS[550].VALUE := 0.0;
   STATUS[550].TRIGVALUE := 0.0;
   STATUS[550].EXT.AlarmWarnUnAck := FALSE;
   STATUS[550].EXT.AckRequired := FALSE;
   STATUS[550].EXT.Maintanence := FALSE;
   STATUS[550].EXT.Operation := FALSE;
   STATUS[550].EXT.Forced := FALSE;
   STATUS[550].EXT.BIT29 := FALSE;
   STATUS[550].EXT.BIT30 := FALSE;
   STATUS[550].EXT.BIT31 := FALSE;
   STATUS[550].EXT.ModeBit1 := FALSE;
   STATUS[550].EXT.ModeBit2 := FALSE;
   STATUS[550].EXT.ModeBit3 := FALSE;
   STATUS[550].EXT.BIT19 := FALSE;
   STATUS[550].EXT.BIT20 := FALSE;
   STATUS[550].EXT.AlarmSuppressed := FALSE;
   STATUS[550].EXT.AlarmPrsent := FALSE;
   STATUS[550].EXT.AlarmFailUnAck := FALSE;
   STATUS[550].Status := 0;
   STATUS[550].TimeStamp := 16#0000;
   STATUS[551].VALUE := 0.0;
   STATUS[551].TRIGVALUE := 0.0;
   STATUS[551].EXT.AlarmWarnUnAck := FALSE;
   STATUS[551].EXT.AckRequired := FALSE;
   STATUS[551].EXT.Maintanence := FALSE;
   STATUS[551].EXT.Operation := FALSE;
   STATUS[551].EXT.Forced := FALSE;
   STATUS[551].EXT.BIT29 := FALSE;
   STATUS[551].EXT.BIT30 := FALSE;
   STATUS[551].EXT.BIT31 := FALSE;
   STATUS[551].EXT.ModeBit1 := FALSE;
   STATUS[551].EXT.ModeBit2 := FALSE;
   STATUS[551].EXT.ModeBit3 := FALSE;
   STATUS[551].EXT.BIT19 := FALSE;
   STATUS[551].EXT.BIT20 := FALSE;
   STATUS[551].EXT.AlarmSuppressed := FALSE;
   STATUS[551].EXT.AlarmPrsent := FALSE;
   STATUS[551].EXT.AlarmFailUnAck := FALSE;
   STATUS[551].Status := 0;
   STATUS[551].TimeStamp := 16#0000;
   STATUS[552].VALUE := 0.0;
   STATUS[552].TRIGVALUE := 0.0;
   STATUS[552].EXT.AlarmWarnUnAck := FALSE;
   STATUS[552].EXT.AckRequired := FALSE;
   STATUS[552].EXT.Maintanence := FALSE;
   STATUS[552].EXT.Operation := FALSE;
   STATUS[552].EXT.Forced := FALSE;
   STATUS[552].EXT.BIT29 := FALSE;
   STATUS[552].EXT.BIT30 := FALSE;
   STATUS[552].EXT.BIT31 := FALSE;
   STATUS[552].EXT.ModeBit1 := FALSE;
   STATUS[552].EXT.ModeBit2 := FALSE;
   STATUS[552].EXT.ModeBit3 := FALSE;
   STATUS[552].EXT.BIT19 := FALSE;
   STATUS[552].EXT.BIT20 := FALSE;
   STATUS[552].EXT.AlarmSuppressed := FALSE;
   STATUS[552].EXT.AlarmPrsent := FALSE;
   STATUS[552].EXT.AlarmFailUnAck := FALSE;
   STATUS[552].Status := 0;
   STATUS[552].TimeStamp := 16#0000;
   STATUS[553].VALUE := 0.0;
   STATUS[553].TRIGVALUE := 0.0;
   STATUS[553].EXT.AlarmWarnUnAck := FALSE;
   STATUS[553].EXT.AckRequired := FALSE;
   STATUS[553].EXT.Maintanence := FALSE;
   STATUS[553].EXT.Operation := FALSE;
   STATUS[553].EXT.Forced := FALSE;
   STATUS[553].EXT.BIT29 := FALSE;
   STATUS[553].EXT.BIT30 := FALSE;
   STATUS[553].EXT.BIT31 := FALSE;
   STATUS[553].EXT.ModeBit1 := FALSE;
   STATUS[553].EXT.ModeBit2 := FALSE;
   STATUS[553].EXT.ModeBit3 := FALSE;
   STATUS[553].EXT.BIT19 := FALSE;
   STATUS[553].EXT.BIT20 := FALSE;
   STATUS[553].EXT.AlarmSuppressed := FALSE;
   STATUS[553].EXT.AlarmPrsent := FALSE;
   STATUS[553].EXT.AlarmFailUnAck := FALSE;
   STATUS[553].Status := 0;
   STATUS[553].TimeStamp := 16#0000;
   STATUS[554].VALUE := 0.0;
   STATUS[554].TRIGVALUE := 0.0;
   STATUS[554].EXT.AlarmWarnUnAck := FALSE;
   STATUS[554].EXT.AckRequired := FALSE;
   STATUS[554].EXT.Maintanence := FALSE;
   STATUS[554].EXT.Operation := FALSE;
   STATUS[554].EXT.Forced := FALSE;
   STATUS[554].EXT.BIT29 := FALSE;
   STATUS[554].EXT.BIT30 := FALSE;
   STATUS[554].EXT.BIT31 := FALSE;
   STATUS[554].EXT.ModeBit1 := FALSE;
   STATUS[554].EXT.ModeBit2 := FALSE;
   STATUS[554].EXT.ModeBit3 := FALSE;
   STATUS[554].EXT.BIT19 := FALSE;
   STATUS[554].EXT.BIT20 := FALSE;
   STATUS[554].EXT.AlarmSuppressed := FALSE;
   STATUS[554].EXT.AlarmPrsent := FALSE;
   STATUS[554].EXT.AlarmFailUnAck := FALSE;
   STATUS[554].Status := 0;
   STATUS[554].TimeStamp := 16#0000;
   STATUS[555].VALUE := 0.0;
   STATUS[555].TRIGVALUE := 0.0;
   STATUS[555].EXT.AlarmWarnUnAck := FALSE;
   STATUS[555].EXT.AckRequired := FALSE;
   STATUS[555].EXT.Maintanence := FALSE;
   STATUS[555].EXT.Operation := FALSE;
   STATUS[555].EXT.Forced := FALSE;
   STATUS[555].EXT.BIT29 := FALSE;
   STATUS[555].EXT.BIT30 := FALSE;
   STATUS[555].EXT.BIT31 := FALSE;
   STATUS[555].EXT.ModeBit1 := FALSE;
   STATUS[555].EXT.ModeBit2 := FALSE;
   STATUS[555].EXT.ModeBit3 := FALSE;
   STATUS[555].EXT.BIT19 := FALSE;
   STATUS[555].EXT.BIT20 := FALSE;
   STATUS[555].EXT.AlarmSuppressed := FALSE;
   STATUS[555].EXT.AlarmPrsent := FALSE;
   STATUS[555].EXT.AlarmFailUnAck := FALSE;
   STATUS[555].Status := 0;
   STATUS[555].TimeStamp := 16#0000;
   STATUS[556].VALUE := 0.0;
   STATUS[556].TRIGVALUE := 0.0;
   STATUS[556].EXT.AlarmWarnUnAck := FALSE;
   STATUS[556].EXT.AckRequired := FALSE;
   STATUS[556].EXT.Maintanence := FALSE;
   STATUS[556].EXT.Operation := FALSE;
   STATUS[556].EXT.Forced := FALSE;
   STATUS[556].EXT.BIT29 := FALSE;
   STATUS[556].EXT.BIT30 := FALSE;
   STATUS[556].EXT.BIT31 := FALSE;
   STATUS[556].EXT.ModeBit1 := FALSE;
   STATUS[556].EXT.ModeBit2 := FALSE;
   STATUS[556].EXT.ModeBit3 := FALSE;
   STATUS[556].EXT.BIT19 := FALSE;
   STATUS[556].EXT.BIT20 := FALSE;
   STATUS[556].EXT.AlarmSuppressed := FALSE;
   STATUS[556].EXT.AlarmPrsent := FALSE;
   STATUS[556].EXT.AlarmFailUnAck := FALSE;
   STATUS[556].Status := 0;
   STATUS[556].TimeStamp := 16#0000;
   STATUS[557].VALUE := 0.0;
   STATUS[557].TRIGVALUE := 0.0;
   STATUS[557].EXT.AlarmWarnUnAck := FALSE;
   STATUS[557].EXT.AckRequired := FALSE;
   STATUS[557].EXT.Maintanence := FALSE;
   STATUS[557].EXT.Operation := FALSE;
   STATUS[557].EXT.Forced := FALSE;
   STATUS[557].EXT.BIT29 := FALSE;
   STATUS[557].EXT.BIT30 := FALSE;
   STATUS[557].EXT.BIT31 := FALSE;
   STATUS[557].EXT.ModeBit1 := FALSE;
   STATUS[557].EXT.ModeBit2 := FALSE;
   STATUS[557].EXT.ModeBit3 := FALSE;
   STATUS[557].EXT.BIT19 := FALSE;
   STATUS[557].EXT.BIT20 := FALSE;
   STATUS[557].EXT.AlarmSuppressed := FALSE;
   STATUS[557].EXT.AlarmPrsent := FALSE;
   STATUS[557].EXT.AlarmFailUnAck := FALSE;
   STATUS[557].Status := 0;
   STATUS[557].TimeStamp := 16#0000;
   STATUS[558].VALUE := 0.0;
   STATUS[558].TRIGVALUE := 0.0;
   STATUS[558].EXT.AlarmWarnUnAck := FALSE;
   STATUS[558].EXT.AckRequired := FALSE;
   STATUS[558].EXT.Maintanence := FALSE;
   STATUS[558].EXT.Operation := FALSE;
   STATUS[558].EXT.Forced := FALSE;
   STATUS[558].EXT.BIT29 := FALSE;
   STATUS[558].EXT.BIT30 := FALSE;
   STATUS[558].EXT.BIT31 := FALSE;
   STATUS[558].EXT.ModeBit1 := FALSE;
   STATUS[558].EXT.ModeBit2 := FALSE;
   STATUS[558].EXT.ModeBit3 := FALSE;
   STATUS[558].EXT.BIT19 := FALSE;
   STATUS[558].EXT.BIT20 := FALSE;
   STATUS[558].EXT.AlarmSuppressed := FALSE;
   STATUS[558].EXT.AlarmPrsent := FALSE;
   STATUS[558].EXT.AlarmFailUnAck := FALSE;
   STATUS[558].Status := 0;
   STATUS[558].TimeStamp := 16#0000;
   STATUS[559].VALUE := 0.0;
   STATUS[559].TRIGVALUE := 0.0;
   STATUS[559].EXT.AlarmWarnUnAck := FALSE;
   STATUS[559].EXT.AckRequired := FALSE;
   STATUS[559].EXT.Maintanence := FALSE;
   STATUS[559].EXT.Operation := FALSE;
   STATUS[559].EXT.Forced := FALSE;
   STATUS[559].EXT.BIT29 := FALSE;
   STATUS[559].EXT.BIT30 := FALSE;
   STATUS[559].EXT.BIT31 := FALSE;
   STATUS[559].EXT.ModeBit1 := FALSE;
   STATUS[559].EXT.ModeBit2 := FALSE;
   STATUS[559].EXT.ModeBit3 := FALSE;
   STATUS[559].EXT.BIT19 := FALSE;
   STATUS[559].EXT.BIT20 := FALSE;
   STATUS[559].EXT.AlarmSuppressed := FALSE;
   STATUS[559].EXT.AlarmPrsent := FALSE;
   STATUS[559].EXT.AlarmFailUnAck := FALSE;
   STATUS[559].Status := 0;
   STATUS[559].TimeStamp := 16#0000;
   STATUS[560].VALUE := 0.0;
   STATUS[560].TRIGVALUE := 0.0;
   STATUS[560].EXT.AlarmWarnUnAck := FALSE;
   STATUS[560].EXT.AckRequired := FALSE;
   STATUS[560].EXT.Maintanence := FALSE;
   STATUS[560].EXT.Operation := FALSE;
   STATUS[560].EXT.Forced := FALSE;
   STATUS[560].EXT.BIT29 := FALSE;
   STATUS[560].EXT.BIT30 := FALSE;
   STATUS[560].EXT.BIT31 := FALSE;
   STATUS[560].EXT.ModeBit1 := FALSE;
   STATUS[560].EXT.ModeBit2 := FALSE;
   STATUS[560].EXT.ModeBit3 := FALSE;
   STATUS[560].EXT.BIT19 := FALSE;
   STATUS[560].EXT.BIT20 := FALSE;
   STATUS[560].EXT.AlarmSuppressed := FALSE;
   STATUS[560].EXT.AlarmPrsent := FALSE;
   STATUS[560].EXT.AlarmFailUnAck := FALSE;
   STATUS[560].Status := 0;
   STATUS[560].TimeStamp := 16#0000;
   STATUS[561].VALUE := 0.0;
   STATUS[561].TRIGVALUE := 0.0;
   STATUS[561].EXT.AlarmWarnUnAck := FALSE;
   STATUS[561].EXT.AckRequired := FALSE;
   STATUS[561].EXT.Maintanence := FALSE;
   STATUS[561].EXT.Operation := FALSE;
   STATUS[561].EXT.Forced := FALSE;
   STATUS[561].EXT.BIT29 := FALSE;
   STATUS[561].EXT.BIT30 := FALSE;
   STATUS[561].EXT.BIT31 := FALSE;
   STATUS[561].EXT.ModeBit1 := FALSE;
   STATUS[561].EXT.ModeBit2 := FALSE;
   STATUS[561].EXT.ModeBit3 := FALSE;
   STATUS[561].EXT.BIT19 := FALSE;
   STATUS[561].EXT.BIT20 := FALSE;
   STATUS[561].EXT.AlarmSuppressed := FALSE;
   STATUS[561].EXT.AlarmPrsent := FALSE;
   STATUS[561].EXT.AlarmFailUnAck := FALSE;
   STATUS[561].Status := 0;
   STATUS[561].TimeStamp := 16#0000;
   STATUS[562].VALUE := 0.0;
   STATUS[562].TRIGVALUE := 0.0;
   STATUS[562].EXT.AlarmWarnUnAck := FALSE;
   STATUS[562].EXT.AckRequired := FALSE;
   STATUS[562].EXT.Maintanence := FALSE;
   STATUS[562].EXT.Operation := FALSE;
   STATUS[562].EXT.Forced := FALSE;
   STATUS[562].EXT.BIT29 := FALSE;
   STATUS[562].EXT.BIT30 := FALSE;
   STATUS[562].EXT.BIT31 := FALSE;
   STATUS[562].EXT.ModeBit1 := FALSE;
   STATUS[562].EXT.ModeBit2 := FALSE;
   STATUS[562].EXT.ModeBit3 := FALSE;
   STATUS[562].EXT.BIT19 := FALSE;
   STATUS[562].EXT.BIT20 := FALSE;
   STATUS[562].EXT.AlarmSuppressed := FALSE;
   STATUS[562].EXT.AlarmPrsent := FALSE;
   STATUS[562].EXT.AlarmFailUnAck := FALSE;
   STATUS[562].Status := 0;
   STATUS[562].TimeStamp := 16#0000;
   STATUS[563].VALUE := 0.0;
   STATUS[563].TRIGVALUE := 0.0;
   STATUS[563].EXT.AlarmWarnUnAck := FALSE;
   STATUS[563].EXT.AckRequired := FALSE;
   STATUS[563].EXT.Maintanence := FALSE;
   STATUS[563].EXT.Operation := FALSE;
   STATUS[563].EXT.Forced := FALSE;
   STATUS[563].EXT.BIT29 := FALSE;
   STATUS[563].EXT.BIT30 := FALSE;
   STATUS[563].EXT.BIT31 := FALSE;
   STATUS[563].EXT.ModeBit1 := FALSE;
   STATUS[563].EXT.ModeBit2 := FALSE;
   STATUS[563].EXT.ModeBit3 := FALSE;
   STATUS[563].EXT.BIT19 := FALSE;
   STATUS[563].EXT.BIT20 := FALSE;
   STATUS[563].EXT.AlarmSuppressed := FALSE;
   STATUS[563].EXT.AlarmPrsent := FALSE;
   STATUS[563].EXT.AlarmFailUnAck := FALSE;
   STATUS[563].Status := 0;
   STATUS[563].TimeStamp := 16#0000;
   STATUS[564].VALUE := 0.0;
   STATUS[564].TRIGVALUE := 0.0;
   STATUS[564].EXT.AlarmWarnUnAck := FALSE;
   STATUS[564].EXT.AckRequired := FALSE;
   STATUS[564].EXT.Maintanence := FALSE;
   STATUS[564].EXT.Operation := FALSE;
   STATUS[564].EXT.Forced := FALSE;
   STATUS[564].EXT.BIT29 := FALSE;
   STATUS[564].EXT.BIT30 := FALSE;
   STATUS[564].EXT.BIT31 := FALSE;
   STATUS[564].EXT.ModeBit1 := FALSE;
   STATUS[564].EXT.ModeBit2 := FALSE;
   STATUS[564].EXT.ModeBit3 := FALSE;
   STATUS[564].EXT.BIT19 := FALSE;
   STATUS[564].EXT.BIT20 := FALSE;
   STATUS[564].EXT.AlarmSuppressed := FALSE;
   STATUS[564].EXT.AlarmPrsent := FALSE;
   STATUS[564].EXT.AlarmFailUnAck := FALSE;
   STATUS[564].Status := 0;
   STATUS[564].TimeStamp := 16#0000;
   STATUS[565].VALUE := 0.0;
   STATUS[565].TRIGVALUE := 0.0;
   STATUS[565].EXT.AlarmWarnUnAck := FALSE;
   STATUS[565].EXT.AckRequired := FALSE;
   STATUS[565].EXT.Maintanence := FALSE;
   STATUS[565].EXT.Operation := FALSE;
   STATUS[565].EXT.Forced := FALSE;
   STATUS[565].EXT.BIT29 := FALSE;
   STATUS[565].EXT.BIT30 := FALSE;
   STATUS[565].EXT.BIT31 := FALSE;
   STATUS[565].EXT.ModeBit1 := FALSE;
   STATUS[565].EXT.ModeBit2 := FALSE;
   STATUS[565].EXT.ModeBit3 := FALSE;
   STATUS[565].EXT.BIT19 := FALSE;
   STATUS[565].EXT.BIT20 := FALSE;
   STATUS[565].EXT.AlarmSuppressed := FALSE;
   STATUS[565].EXT.AlarmPrsent := FALSE;
   STATUS[565].EXT.AlarmFailUnAck := FALSE;
   STATUS[565].Status := 0;
   STATUS[565].TimeStamp := 16#0000;
   STATUS[566].VALUE := 0.0;
   STATUS[566].TRIGVALUE := 0.0;
   STATUS[566].EXT.AlarmWarnUnAck := FALSE;
   STATUS[566].EXT.AckRequired := FALSE;
   STATUS[566].EXT.Maintanence := FALSE;
   STATUS[566].EXT.Operation := FALSE;
   STATUS[566].EXT.Forced := FALSE;
   STATUS[566].EXT.BIT29 := FALSE;
   STATUS[566].EXT.BIT30 := FALSE;
   STATUS[566].EXT.BIT31 := FALSE;
   STATUS[566].EXT.ModeBit1 := FALSE;
   STATUS[566].EXT.ModeBit2 := FALSE;
   STATUS[566].EXT.ModeBit3 := FALSE;
   STATUS[566].EXT.BIT19 := FALSE;
   STATUS[566].EXT.BIT20 := FALSE;
   STATUS[566].EXT.AlarmSuppressed := FALSE;
   STATUS[566].EXT.AlarmPrsent := FALSE;
   STATUS[566].EXT.AlarmFailUnAck := FALSE;
   STATUS[566].Status := 0;
   STATUS[566].TimeStamp := 16#0000;
   STATUS[567].VALUE := 0.0;
   STATUS[567].TRIGVALUE := 0.0;
   STATUS[567].EXT.AlarmWarnUnAck := FALSE;
   STATUS[567].EXT.AckRequired := FALSE;
   STATUS[567].EXT.Maintanence := FALSE;
   STATUS[567].EXT.Operation := FALSE;
   STATUS[567].EXT.Forced := FALSE;
   STATUS[567].EXT.BIT29 := FALSE;
   STATUS[567].EXT.BIT30 := FALSE;
   STATUS[567].EXT.BIT31 := FALSE;
   STATUS[567].EXT.ModeBit1 := FALSE;
   STATUS[567].EXT.ModeBit2 := FALSE;
   STATUS[567].EXT.ModeBit3 := FALSE;
   STATUS[567].EXT.BIT19 := FALSE;
   STATUS[567].EXT.BIT20 := FALSE;
   STATUS[567].EXT.AlarmSuppressed := FALSE;
   STATUS[567].EXT.AlarmPrsent := FALSE;
   STATUS[567].EXT.AlarmFailUnAck := FALSE;
   STATUS[567].Status := 0;
   STATUS[567].TimeStamp := 16#0000;
   STATUS[568].VALUE := 0.0;
   STATUS[568].TRIGVALUE := 0.0;
   STATUS[568].EXT.AlarmWarnUnAck := FALSE;
   STATUS[568].EXT.AckRequired := FALSE;
   STATUS[568].EXT.Maintanence := FALSE;
   STATUS[568].EXT.Operation := FALSE;
   STATUS[568].EXT.Forced := FALSE;
   STATUS[568].EXT.BIT29 := FALSE;
   STATUS[568].EXT.BIT30 := FALSE;
   STATUS[568].EXT.BIT31 := FALSE;
   STATUS[568].EXT.ModeBit1 := FALSE;
   STATUS[568].EXT.ModeBit2 := FALSE;
   STATUS[568].EXT.ModeBit3 := FALSE;
   STATUS[568].EXT.BIT19 := FALSE;
   STATUS[568].EXT.BIT20 := FALSE;
   STATUS[568].EXT.AlarmSuppressed := FALSE;
   STATUS[568].EXT.AlarmPrsent := FALSE;
   STATUS[568].EXT.AlarmFailUnAck := FALSE;
   STATUS[568].Status := 0;
   STATUS[568].TimeStamp := 16#0000;
   STATUS[569].VALUE := 0.0;
   STATUS[569].TRIGVALUE := 0.0;
   STATUS[569].EXT.AlarmWarnUnAck := FALSE;
   STATUS[569].EXT.AckRequired := FALSE;
   STATUS[569].EXT.Maintanence := FALSE;
   STATUS[569].EXT.Operation := FALSE;
   STATUS[569].EXT.Forced := FALSE;
   STATUS[569].EXT.BIT29 := FALSE;
   STATUS[569].EXT.BIT30 := FALSE;
   STATUS[569].EXT.BIT31 := FALSE;
   STATUS[569].EXT.ModeBit1 := FALSE;
   STATUS[569].EXT.ModeBit2 := FALSE;
   STATUS[569].EXT.ModeBit3 := FALSE;
   STATUS[569].EXT.BIT19 := FALSE;
   STATUS[569].EXT.BIT20 := FALSE;
   STATUS[569].EXT.AlarmSuppressed := FALSE;
   STATUS[569].EXT.AlarmPrsent := FALSE;
   STATUS[569].EXT.AlarmFailUnAck := FALSE;
   STATUS[569].Status := 0;
   STATUS[569].TimeStamp := 16#0000;
   STATUS[570].VALUE := 0.0;
   STATUS[570].TRIGVALUE := 0.0;
   STATUS[570].EXT.AlarmWarnUnAck := FALSE;
   STATUS[570].EXT.AckRequired := FALSE;
   STATUS[570].EXT.Maintanence := FALSE;
   STATUS[570].EXT.Operation := FALSE;
   STATUS[570].EXT.Forced := FALSE;
   STATUS[570].EXT.BIT29 := FALSE;
   STATUS[570].EXT.BIT30 := FALSE;
   STATUS[570].EXT.BIT31 := FALSE;
   STATUS[570].EXT.ModeBit1 := FALSE;
   STATUS[570].EXT.ModeBit2 := FALSE;
   STATUS[570].EXT.ModeBit3 := FALSE;
   STATUS[570].EXT.BIT19 := FALSE;
   STATUS[570].EXT.BIT20 := FALSE;
   STATUS[570].EXT.AlarmSuppressed := FALSE;
   STATUS[570].EXT.AlarmPrsent := FALSE;
   STATUS[570].EXT.AlarmFailUnAck := FALSE;
   STATUS[570].Status := 0;
   STATUS[570].TimeStamp := 16#0000;
   STATUS[571].VALUE := 0.0;
   STATUS[571].TRIGVALUE := 0.0;
   STATUS[571].EXT.AlarmWarnUnAck := FALSE;
   STATUS[571].EXT.AckRequired := FALSE;
   STATUS[571].EXT.Maintanence := FALSE;
   STATUS[571].EXT.Operation := FALSE;
   STATUS[571].EXT.Forced := FALSE;
   STATUS[571].EXT.BIT29 := FALSE;
   STATUS[571].EXT.BIT30 := FALSE;
   STATUS[571].EXT.BIT31 := FALSE;
   STATUS[571].EXT.ModeBit1 := FALSE;
   STATUS[571].EXT.ModeBit2 := FALSE;
   STATUS[571].EXT.ModeBit3 := FALSE;
   STATUS[571].EXT.BIT19 := FALSE;
   STATUS[571].EXT.BIT20 := FALSE;
   STATUS[571].EXT.AlarmSuppressed := FALSE;
   STATUS[571].EXT.AlarmPrsent := FALSE;
   STATUS[571].EXT.AlarmFailUnAck := FALSE;
   STATUS[571].Status := 0;
   STATUS[571].TimeStamp := 16#0000;
   STATUS[572].VALUE := 0.0;
   STATUS[572].TRIGVALUE := 0.0;
   STATUS[572].EXT.AlarmWarnUnAck := FALSE;
   STATUS[572].EXT.AckRequired := FALSE;
   STATUS[572].EXT.Maintanence := FALSE;
   STATUS[572].EXT.Operation := FALSE;
   STATUS[572].EXT.Forced := FALSE;
   STATUS[572].EXT.BIT29 := FALSE;
   STATUS[572].EXT.BIT30 := FALSE;
   STATUS[572].EXT.BIT31 := FALSE;
   STATUS[572].EXT.ModeBit1 := FALSE;
   STATUS[572].EXT.ModeBit2 := FALSE;
   STATUS[572].EXT.ModeBit3 := FALSE;
   STATUS[572].EXT.BIT19 := FALSE;
   STATUS[572].EXT.BIT20 := FALSE;
   STATUS[572].EXT.AlarmSuppressed := FALSE;
   STATUS[572].EXT.AlarmPrsent := FALSE;
   STATUS[572].EXT.AlarmFailUnAck := FALSE;
   STATUS[572].Status := 0;
   STATUS[572].TimeStamp := 16#0000;
   STATUS[573].VALUE := 0.0;
   STATUS[573].TRIGVALUE := 0.0;
   STATUS[573].EXT.AlarmWarnUnAck := FALSE;
   STATUS[573].EXT.AckRequired := FALSE;
   STATUS[573].EXT.Maintanence := FALSE;
   STATUS[573].EXT.Operation := FALSE;
   STATUS[573].EXT.Forced := FALSE;
   STATUS[573].EXT.BIT29 := FALSE;
   STATUS[573].EXT.BIT30 := FALSE;
   STATUS[573].EXT.BIT31 := FALSE;
   STATUS[573].EXT.ModeBit1 := FALSE;
   STATUS[573].EXT.ModeBit2 := FALSE;
   STATUS[573].EXT.ModeBit3 := FALSE;
   STATUS[573].EXT.BIT19 := FALSE;
   STATUS[573].EXT.BIT20 := FALSE;
   STATUS[573].EXT.AlarmSuppressed := FALSE;
   STATUS[573].EXT.AlarmPrsent := FALSE;
   STATUS[573].EXT.AlarmFailUnAck := FALSE;
   STATUS[573].Status := 0;
   STATUS[573].TimeStamp := 16#0000;
   STATUS[574].VALUE := 0.0;
   STATUS[574].TRIGVALUE := 0.0;
   STATUS[574].EXT.AlarmWarnUnAck := FALSE;
   STATUS[574].EXT.AckRequired := FALSE;
   STATUS[574].EXT.Maintanence := FALSE;
   STATUS[574].EXT.Operation := FALSE;
   STATUS[574].EXT.Forced := FALSE;
   STATUS[574].EXT.BIT29 := FALSE;
   STATUS[574].EXT.BIT30 := FALSE;
   STATUS[574].EXT.BIT31 := FALSE;
   STATUS[574].EXT.ModeBit1 := FALSE;
   STATUS[574].EXT.ModeBit2 := FALSE;
   STATUS[574].EXT.ModeBit3 := FALSE;
   STATUS[574].EXT.BIT19 := FALSE;
   STATUS[574].EXT.BIT20 := FALSE;
   STATUS[574].EXT.AlarmSuppressed := FALSE;
   STATUS[574].EXT.AlarmPrsent := FALSE;
   STATUS[574].EXT.AlarmFailUnAck := FALSE;
   STATUS[574].Status := 0;
   STATUS[574].TimeStamp := 16#0000;
   STATUS[575].VALUE := 0.0;
   STATUS[575].TRIGVALUE := 0.0;
   STATUS[575].EXT.AlarmWarnUnAck := FALSE;
   STATUS[575].EXT.AckRequired := FALSE;
   STATUS[575].EXT.Maintanence := FALSE;
   STATUS[575].EXT.Operation := FALSE;
   STATUS[575].EXT.Forced := FALSE;
   STATUS[575].EXT.BIT29 := FALSE;
   STATUS[575].EXT.BIT30 := FALSE;
   STATUS[575].EXT.BIT31 := FALSE;
   STATUS[575].EXT.ModeBit1 := FALSE;
   STATUS[575].EXT.ModeBit2 := FALSE;
   STATUS[575].EXT.ModeBit3 := FALSE;
   STATUS[575].EXT.BIT19 := FALSE;
   STATUS[575].EXT.BIT20 := FALSE;
   STATUS[575].EXT.AlarmSuppressed := FALSE;
   STATUS[575].EXT.AlarmPrsent := FALSE;
   STATUS[575].EXT.AlarmFailUnAck := FALSE;
   STATUS[575].Status := 0;
   STATUS[575].TimeStamp := 16#0000;
   STATUS[576].VALUE := 0.0;
   STATUS[576].TRIGVALUE := 0.0;
   STATUS[576].EXT.AlarmWarnUnAck := FALSE;
   STATUS[576].EXT.AckRequired := FALSE;
   STATUS[576].EXT.Maintanence := FALSE;
   STATUS[576].EXT.Operation := FALSE;
   STATUS[576].EXT.Forced := FALSE;
   STATUS[576].EXT.BIT29 := FALSE;
   STATUS[576].EXT.BIT30 := FALSE;
   STATUS[576].EXT.BIT31 := FALSE;
   STATUS[576].EXT.ModeBit1 := FALSE;
   STATUS[576].EXT.ModeBit2 := FALSE;
   STATUS[576].EXT.ModeBit3 := FALSE;
   STATUS[576].EXT.BIT19 := FALSE;
   STATUS[576].EXT.BIT20 := FALSE;
   STATUS[576].EXT.AlarmSuppressed := FALSE;
   STATUS[576].EXT.AlarmPrsent := FALSE;
   STATUS[576].EXT.AlarmFailUnAck := FALSE;
   STATUS[576].Status := 0;
   STATUS[576].TimeStamp := 16#0000;
   STATUS[577].VALUE := 0.0;
   STATUS[577].TRIGVALUE := 0.0;
   STATUS[577].EXT.AlarmWarnUnAck := FALSE;
   STATUS[577].EXT.AckRequired := FALSE;
   STATUS[577].EXT.Maintanence := FALSE;
   STATUS[577].EXT.Operation := FALSE;
   STATUS[577].EXT.Forced := FALSE;
   STATUS[577].EXT.BIT29 := FALSE;
   STATUS[577].EXT.BIT30 := FALSE;
   STATUS[577].EXT.BIT31 := FALSE;
   STATUS[577].EXT.ModeBit1 := FALSE;
   STATUS[577].EXT.ModeBit2 := FALSE;
   STATUS[577].EXT.ModeBit3 := FALSE;
   STATUS[577].EXT.BIT19 := FALSE;
   STATUS[577].EXT.BIT20 := FALSE;
   STATUS[577].EXT.AlarmSuppressed := FALSE;
   STATUS[577].EXT.AlarmPrsent := FALSE;
   STATUS[577].EXT.AlarmFailUnAck := FALSE;
   STATUS[577].Status := 0;
   STATUS[577].TimeStamp := 16#0000;
   STATUS[578].VALUE := 0.0;
   STATUS[578].TRIGVALUE := 0.0;
   STATUS[578].EXT.AlarmWarnUnAck := FALSE;
   STATUS[578].EXT.AckRequired := FALSE;
   STATUS[578].EXT.Maintanence := FALSE;
   STATUS[578].EXT.Operation := FALSE;
   STATUS[578].EXT.Forced := FALSE;
   STATUS[578].EXT.BIT29 := FALSE;
   STATUS[578].EXT.BIT30 := FALSE;
   STATUS[578].EXT.BIT31 := FALSE;
   STATUS[578].EXT.ModeBit1 := FALSE;
   STATUS[578].EXT.ModeBit2 := FALSE;
   STATUS[578].EXT.ModeBit3 := FALSE;
   STATUS[578].EXT.BIT19 := FALSE;
   STATUS[578].EXT.BIT20 := FALSE;
   STATUS[578].EXT.AlarmSuppressed := FALSE;
   STATUS[578].EXT.AlarmPrsent := FALSE;
   STATUS[578].EXT.AlarmFailUnAck := FALSE;
   STATUS[578].Status := 0;
   STATUS[578].TimeStamp := 16#0000;
   STATUS[579].VALUE := 0.0;
   STATUS[579].TRIGVALUE := 0.0;
   STATUS[579].EXT.AlarmWarnUnAck := FALSE;
   STATUS[579].EXT.AckRequired := FALSE;
   STATUS[579].EXT.Maintanence := FALSE;
   STATUS[579].EXT.Operation := FALSE;
   STATUS[579].EXT.Forced := FALSE;
   STATUS[579].EXT.BIT29 := FALSE;
   STATUS[579].EXT.BIT30 := FALSE;
   STATUS[579].EXT.BIT31 := FALSE;
   STATUS[579].EXT.ModeBit1 := FALSE;
   STATUS[579].EXT.ModeBit2 := FALSE;
   STATUS[579].EXT.ModeBit3 := FALSE;
   STATUS[579].EXT.BIT19 := FALSE;
   STATUS[579].EXT.BIT20 := FALSE;
   STATUS[579].EXT.AlarmSuppressed := FALSE;
   STATUS[579].EXT.AlarmPrsent := FALSE;
   STATUS[579].EXT.AlarmFailUnAck := FALSE;
   STATUS[579].Status := 0;
   STATUS[579].TimeStamp := 16#0000;
   STATUS[580].VALUE := 0.0;
   STATUS[580].TRIGVALUE := 0.0;
   STATUS[580].EXT.AlarmWarnUnAck := FALSE;
   STATUS[580].EXT.AckRequired := FALSE;
   STATUS[580].EXT.Maintanence := FALSE;
   STATUS[580].EXT.Operation := FALSE;
   STATUS[580].EXT.Forced := FALSE;
   STATUS[580].EXT.BIT29 := FALSE;
   STATUS[580].EXT.BIT30 := FALSE;
   STATUS[580].EXT.BIT31 := FALSE;
   STATUS[580].EXT.ModeBit1 := FALSE;
   STATUS[580].EXT.ModeBit2 := FALSE;
   STATUS[580].EXT.ModeBit3 := FALSE;
   STATUS[580].EXT.BIT19 := FALSE;
   STATUS[580].EXT.BIT20 := FALSE;
   STATUS[580].EXT.AlarmSuppressed := FALSE;
   STATUS[580].EXT.AlarmPrsent := FALSE;
   STATUS[580].EXT.AlarmFailUnAck := FALSE;
   STATUS[580].Status := 0;
   STATUS[580].TimeStamp := 16#0000;
   STATUS[581].VALUE := 0.0;
   STATUS[581].TRIGVALUE := 0.0;
   STATUS[581].EXT.AlarmWarnUnAck := FALSE;
   STATUS[581].EXT.AckRequired := FALSE;
   STATUS[581].EXT.Maintanence := FALSE;
   STATUS[581].EXT.Operation := FALSE;
   STATUS[581].EXT.Forced := FALSE;
   STATUS[581].EXT.BIT29 := FALSE;
   STATUS[581].EXT.BIT30 := FALSE;
   STATUS[581].EXT.BIT31 := FALSE;
   STATUS[581].EXT.ModeBit1 := FALSE;
   STATUS[581].EXT.ModeBit2 := FALSE;
   STATUS[581].EXT.ModeBit3 := FALSE;
   STATUS[581].EXT.BIT19 := FALSE;
   STATUS[581].EXT.BIT20 := FALSE;
   STATUS[581].EXT.AlarmSuppressed := FALSE;
   STATUS[581].EXT.AlarmPrsent := FALSE;
   STATUS[581].EXT.AlarmFailUnAck := FALSE;
   STATUS[581].Status := 0;
   STATUS[581].TimeStamp := 16#0000;
   STATUS[582].VALUE := 0.0;
   STATUS[582].TRIGVALUE := 0.0;
   STATUS[582].EXT.AlarmWarnUnAck := FALSE;
   STATUS[582].EXT.AckRequired := FALSE;
   STATUS[582].EXT.Maintanence := FALSE;
   STATUS[582].EXT.Operation := FALSE;
   STATUS[582].EXT.Forced := FALSE;
   STATUS[582].EXT.BIT29 := FALSE;
   STATUS[582].EXT.BIT30 := FALSE;
   STATUS[582].EXT.BIT31 := FALSE;
   STATUS[582].EXT.ModeBit1 := FALSE;
   STATUS[582].EXT.ModeBit2 := FALSE;
   STATUS[582].EXT.ModeBit3 := FALSE;
   STATUS[582].EXT.BIT19 := FALSE;
   STATUS[582].EXT.BIT20 := FALSE;
   STATUS[582].EXT.AlarmSuppressed := FALSE;
   STATUS[582].EXT.AlarmPrsent := FALSE;
   STATUS[582].EXT.AlarmFailUnAck := FALSE;
   STATUS[582].Status := 0;
   STATUS[582].TimeStamp := 16#0000;
   STATUS[583].VALUE := 0.0;
   STATUS[583].TRIGVALUE := 0.0;
   STATUS[583].EXT.AlarmWarnUnAck := FALSE;
   STATUS[583].EXT.AckRequired := FALSE;
   STATUS[583].EXT.Maintanence := FALSE;
   STATUS[583].EXT.Operation := FALSE;
   STATUS[583].EXT.Forced := FALSE;
   STATUS[583].EXT.BIT29 := FALSE;
   STATUS[583].EXT.BIT30 := FALSE;
   STATUS[583].EXT.BIT31 := FALSE;
   STATUS[583].EXT.ModeBit1 := FALSE;
   STATUS[583].EXT.ModeBit2 := FALSE;
   STATUS[583].EXT.ModeBit3 := FALSE;
   STATUS[583].EXT.BIT19 := FALSE;
   STATUS[583].EXT.BIT20 := FALSE;
   STATUS[583].EXT.AlarmSuppressed := FALSE;
   STATUS[583].EXT.AlarmPrsent := FALSE;
   STATUS[583].EXT.AlarmFailUnAck := FALSE;
   STATUS[583].Status := 0;
   STATUS[583].TimeStamp := 16#0000;
   STATUS[584].VALUE := 0.0;
   STATUS[584].TRIGVALUE := 0.0;
   STATUS[584].EXT.AlarmWarnUnAck := FALSE;
   STATUS[584].EXT.AckRequired := FALSE;
   STATUS[584].EXT.Maintanence := FALSE;
   STATUS[584].EXT.Operation := FALSE;
   STATUS[584].EXT.Forced := FALSE;
   STATUS[584].EXT.BIT29 := FALSE;
   STATUS[584].EXT.BIT30 := FALSE;
   STATUS[584].EXT.BIT31 := FALSE;
   STATUS[584].EXT.ModeBit1 := FALSE;
   STATUS[584].EXT.ModeBit2 := FALSE;
   STATUS[584].EXT.ModeBit3 := FALSE;
   STATUS[584].EXT.BIT19 := FALSE;
   STATUS[584].EXT.BIT20 := FALSE;
   STATUS[584].EXT.AlarmSuppressed := FALSE;
   STATUS[584].EXT.AlarmPrsent := FALSE;
   STATUS[584].EXT.AlarmFailUnAck := FALSE;
   STATUS[584].Status := 0;
   STATUS[584].TimeStamp := 16#0000;
   STATUS[585].VALUE := 0.0;
   STATUS[585].TRIGVALUE := 0.0;
   STATUS[585].EXT.AlarmWarnUnAck := FALSE;
   STATUS[585].EXT.AckRequired := FALSE;
   STATUS[585].EXT.Maintanence := FALSE;
   STATUS[585].EXT.Operation := FALSE;
   STATUS[585].EXT.Forced := FALSE;
   STATUS[585].EXT.BIT29 := FALSE;
   STATUS[585].EXT.BIT30 := FALSE;
   STATUS[585].EXT.BIT31 := FALSE;
   STATUS[585].EXT.ModeBit1 := FALSE;
   STATUS[585].EXT.ModeBit2 := FALSE;
   STATUS[585].EXT.ModeBit3 := FALSE;
   STATUS[585].EXT.BIT19 := FALSE;
   STATUS[585].EXT.BIT20 := FALSE;
   STATUS[585].EXT.AlarmSuppressed := FALSE;
   STATUS[585].EXT.AlarmPrsent := FALSE;
   STATUS[585].EXT.AlarmFailUnAck := FALSE;
   STATUS[585].Status := 0;
   STATUS[585].TimeStamp := 16#0000;
   STATUS[586].VALUE := 0.0;
   STATUS[586].TRIGVALUE := 0.0;
   STATUS[586].EXT.AlarmWarnUnAck := FALSE;
   STATUS[586].EXT.AckRequired := FALSE;
   STATUS[586].EXT.Maintanence := FALSE;
   STATUS[586].EXT.Operation := FALSE;
   STATUS[586].EXT.Forced := FALSE;
   STATUS[586].EXT.BIT29 := FALSE;
   STATUS[586].EXT.BIT30 := FALSE;
   STATUS[586].EXT.BIT31 := FALSE;
   STATUS[586].EXT.ModeBit1 := FALSE;
   STATUS[586].EXT.ModeBit2 := FALSE;
   STATUS[586].EXT.ModeBit3 := FALSE;
   STATUS[586].EXT.BIT19 := FALSE;
   STATUS[586].EXT.BIT20 := FALSE;
   STATUS[586].EXT.AlarmSuppressed := FALSE;
   STATUS[586].EXT.AlarmPrsent := FALSE;
   STATUS[586].EXT.AlarmFailUnAck := FALSE;
   STATUS[586].Status := 0;
   STATUS[586].TimeStamp := 16#0000;
   STATUS[587].VALUE := 0.0;
   STATUS[587].TRIGVALUE := 0.0;
   STATUS[587].EXT.AlarmWarnUnAck := FALSE;
   STATUS[587].EXT.AckRequired := FALSE;
   STATUS[587].EXT.Maintanence := FALSE;
   STATUS[587].EXT.Operation := FALSE;
   STATUS[587].EXT.Forced := FALSE;
   STATUS[587].EXT.BIT29 := FALSE;
   STATUS[587].EXT.BIT30 := FALSE;
   STATUS[587].EXT.BIT31 := FALSE;
   STATUS[587].EXT.ModeBit1 := FALSE;
   STATUS[587].EXT.ModeBit2 := FALSE;
   STATUS[587].EXT.ModeBit3 := FALSE;
   STATUS[587].EXT.BIT19 := FALSE;
   STATUS[587].EXT.BIT20 := FALSE;
   STATUS[587].EXT.AlarmSuppressed := FALSE;
   STATUS[587].EXT.AlarmPrsent := FALSE;
   STATUS[587].EXT.AlarmFailUnAck := FALSE;
   STATUS[587].Status := 0;
   STATUS[587].TimeStamp := 16#0000;
   STATUS[588].VALUE := 0.0;
   STATUS[588].TRIGVALUE := 0.0;
   STATUS[588].EXT.AlarmWarnUnAck := FALSE;
   STATUS[588].EXT.AckRequired := FALSE;
   STATUS[588].EXT.Maintanence := FALSE;
   STATUS[588].EXT.Operation := FALSE;
   STATUS[588].EXT.Forced := FALSE;
   STATUS[588].EXT.BIT29 := FALSE;
   STATUS[588].EXT.BIT30 := FALSE;
   STATUS[588].EXT.BIT31 := FALSE;
   STATUS[588].EXT.ModeBit1 := FALSE;
   STATUS[588].EXT.ModeBit2 := FALSE;
   STATUS[588].EXT.ModeBit3 := FALSE;
   STATUS[588].EXT.BIT19 := FALSE;
   STATUS[588].EXT.BIT20 := FALSE;
   STATUS[588].EXT.AlarmSuppressed := FALSE;
   STATUS[588].EXT.AlarmPrsent := FALSE;
   STATUS[588].EXT.AlarmFailUnAck := FALSE;
   STATUS[588].Status := 0;
   STATUS[588].TimeStamp := 16#0000;
   STATUS[589].VALUE := 0.0;
   STATUS[589].TRIGVALUE := 0.0;
   STATUS[589].EXT.AlarmWarnUnAck := FALSE;
   STATUS[589].EXT.AckRequired := FALSE;
   STATUS[589].EXT.Maintanence := FALSE;
   STATUS[589].EXT.Operation := FALSE;
   STATUS[589].EXT.Forced := FALSE;
   STATUS[589].EXT.BIT29 := FALSE;
   STATUS[589].EXT.BIT30 := FALSE;
   STATUS[589].EXT.BIT31 := FALSE;
   STATUS[589].EXT.ModeBit1 := FALSE;
   STATUS[589].EXT.ModeBit2 := FALSE;
   STATUS[589].EXT.ModeBit3 := FALSE;
   STATUS[589].EXT.BIT19 := FALSE;
   STATUS[589].EXT.BIT20 := FALSE;
   STATUS[589].EXT.AlarmSuppressed := FALSE;
   STATUS[589].EXT.AlarmPrsent := FALSE;
   STATUS[589].EXT.AlarmFailUnAck := FALSE;
   STATUS[589].Status := 0;
   STATUS[589].TimeStamp := 16#0000;
   STATUS[590].VALUE := 0.0;
   STATUS[590].TRIGVALUE := 0.0;
   STATUS[590].EXT.AlarmWarnUnAck := FALSE;
   STATUS[590].EXT.AckRequired := FALSE;
   STATUS[590].EXT.Maintanence := FALSE;
   STATUS[590].EXT.Operation := FALSE;
   STATUS[590].EXT.Forced := FALSE;
   STATUS[590].EXT.BIT29 := FALSE;
   STATUS[590].EXT.BIT30 := FALSE;
   STATUS[590].EXT.BIT31 := FALSE;
   STATUS[590].EXT.ModeBit1 := FALSE;
   STATUS[590].EXT.ModeBit2 := FALSE;
   STATUS[590].EXT.ModeBit3 := FALSE;
   STATUS[590].EXT.BIT19 := FALSE;
   STATUS[590].EXT.BIT20 := FALSE;
   STATUS[590].EXT.AlarmSuppressed := FALSE;
   STATUS[590].EXT.AlarmPrsent := FALSE;
   STATUS[590].EXT.AlarmFailUnAck := FALSE;
   STATUS[590].Status := 0;
   STATUS[590].TimeStamp := 16#0000;
   STATUS[591].VALUE := 0.0;
   STATUS[591].TRIGVALUE := 0.0;
   STATUS[591].EXT.AlarmWarnUnAck := FALSE;
   STATUS[591].EXT.AckRequired := FALSE;
   STATUS[591].EXT.Maintanence := FALSE;
   STATUS[591].EXT.Operation := FALSE;
   STATUS[591].EXT.Forced := FALSE;
   STATUS[591].EXT.BIT29 := FALSE;
   STATUS[591].EXT.BIT30 := FALSE;
   STATUS[591].EXT.BIT31 := FALSE;
   STATUS[591].EXT.ModeBit1 := FALSE;
   STATUS[591].EXT.ModeBit2 := FALSE;
   STATUS[591].EXT.ModeBit3 := FALSE;
   STATUS[591].EXT.BIT19 := FALSE;
   STATUS[591].EXT.BIT20 := FALSE;
   STATUS[591].EXT.AlarmSuppressed := FALSE;
   STATUS[591].EXT.AlarmPrsent := FALSE;
   STATUS[591].EXT.AlarmFailUnAck := FALSE;
   STATUS[591].Status := 0;
   STATUS[591].TimeStamp := 16#0000;
   STATUS[592].VALUE := 0.0;
   STATUS[592].TRIGVALUE := 0.0;
   STATUS[592].EXT.AlarmWarnUnAck := FALSE;
   STATUS[592].EXT.AckRequired := FALSE;
   STATUS[592].EXT.Maintanence := FALSE;
   STATUS[592].EXT.Operation := FALSE;
   STATUS[592].EXT.Forced := FALSE;
   STATUS[592].EXT.BIT29 := FALSE;
   STATUS[592].EXT.BIT30 := FALSE;
   STATUS[592].EXT.BIT31 := FALSE;
   STATUS[592].EXT.ModeBit1 := FALSE;
   STATUS[592].EXT.ModeBit2 := FALSE;
   STATUS[592].EXT.ModeBit3 := FALSE;
   STATUS[592].EXT.BIT19 := FALSE;
   STATUS[592].EXT.BIT20 := FALSE;
   STATUS[592].EXT.AlarmSuppressed := FALSE;
   STATUS[592].EXT.AlarmPrsent := FALSE;
   STATUS[592].EXT.AlarmFailUnAck := FALSE;
   STATUS[592].Status := 0;
   STATUS[592].TimeStamp := 16#0000;
   STATUS[593].VALUE := 0.0;
   STATUS[593].TRIGVALUE := 0.0;
   STATUS[593].EXT.AlarmWarnUnAck := FALSE;
   STATUS[593].EXT.AckRequired := FALSE;
   STATUS[593].EXT.Maintanence := FALSE;
   STATUS[593].EXT.Operation := FALSE;
   STATUS[593].EXT.Forced := FALSE;
   STATUS[593].EXT.BIT29 := FALSE;
   STATUS[593].EXT.BIT30 := FALSE;
   STATUS[593].EXT.BIT31 := FALSE;
   STATUS[593].EXT.ModeBit1 := FALSE;
   STATUS[593].EXT.ModeBit2 := FALSE;
   STATUS[593].EXT.ModeBit3 := FALSE;
   STATUS[593].EXT.BIT19 := FALSE;
   STATUS[593].EXT.BIT20 := FALSE;
   STATUS[593].EXT.AlarmSuppressed := FALSE;
   STATUS[593].EXT.AlarmPrsent := FALSE;
   STATUS[593].EXT.AlarmFailUnAck := FALSE;
   STATUS[593].Status := 0;
   STATUS[593].TimeStamp := 16#0000;
   STATUS[594].VALUE := 0.0;
   STATUS[594].TRIGVALUE := 0.0;
   STATUS[594].EXT.AlarmWarnUnAck := FALSE;
   STATUS[594].EXT.AckRequired := FALSE;
   STATUS[594].EXT.Maintanence := FALSE;
   STATUS[594].EXT.Operation := FALSE;
   STATUS[594].EXT.Forced := FALSE;
   STATUS[594].EXT.BIT29 := FALSE;
   STATUS[594].EXT.BIT30 := FALSE;
   STATUS[594].EXT.BIT31 := FALSE;
   STATUS[594].EXT.ModeBit1 := FALSE;
   STATUS[594].EXT.ModeBit2 := FALSE;
   STATUS[594].EXT.ModeBit3 := FALSE;
   STATUS[594].EXT.BIT19 := FALSE;
   STATUS[594].EXT.BIT20 := FALSE;
   STATUS[594].EXT.AlarmSuppressed := FALSE;
   STATUS[594].EXT.AlarmPrsent := FALSE;
   STATUS[594].EXT.AlarmFailUnAck := FALSE;
   STATUS[594].Status := 0;
   STATUS[594].TimeStamp := 16#0000;
   STATUS[595].VALUE := 0.0;
   STATUS[595].TRIGVALUE := 0.0;
   STATUS[595].EXT.AlarmWarnUnAck := FALSE;
   STATUS[595].EXT.AckRequired := FALSE;
   STATUS[595].EXT.Maintanence := FALSE;
   STATUS[595].EXT.Operation := FALSE;
   STATUS[595].EXT.Forced := FALSE;
   STATUS[595].EXT.BIT29 := FALSE;
   STATUS[595].EXT.BIT30 := FALSE;
   STATUS[595].EXT.BIT31 := FALSE;
   STATUS[595].EXT.ModeBit1 := FALSE;
   STATUS[595].EXT.ModeBit2 := FALSE;
   STATUS[595].EXT.ModeBit3 := FALSE;
   STATUS[595].EXT.BIT19 := FALSE;
   STATUS[595].EXT.BIT20 := FALSE;
   STATUS[595].EXT.AlarmSuppressed := FALSE;
   STATUS[595].EXT.AlarmPrsent := FALSE;
   STATUS[595].EXT.AlarmFailUnAck := FALSE;
   STATUS[595].Status := 0;
   STATUS[595].TimeStamp := 16#0000;
   STATUS[596].VALUE := 0.0;
   STATUS[596].TRIGVALUE := 0.0;
   STATUS[596].EXT.AlarmWarnUnAck := FALSE;
   STATUS[596].EXT.AckRequired := FALSE;
   STATUS[596].EXT.Maintanence := FALSE;
   STATUS[596].EXT.Operation := FALSE;
   STATUS[596].EXT.Forced := FALSE;
   STATUS[596].EXT.BIT29 := FALSE;
   STATUS[596].EXT.BIT30 := FALSE;
   STATUS[596].EXT.BIT31 := FALSE;
   STATUS[596].EXT.ModeBit1 := FALSE;
   STATUS[596].EXT.ModeBit2 := FALSE;
   STATUS[596].EXT.ModeBit3 := FALSE;
   STATUS[596].EXT.BIT19 := FALSE;
   STATUS[596].EXT.BIT20 := FALSE;
   STATUS[596].EXT.AlarmSuppressed := FALSE;
   STATUS[596].EXT.AlarmPrsent := FALSE;
   STATUS[596].EXT.AlarmFailUnAck := FALSE;
   STATUS[596].Status := 0;
   STATUS[596].TimeStamp := 16#0000;
   STATUS[597].VALUE := 0.0;
   STATUS[597].TRIGVALUE := 0.0;
   STATUS[597].EXT.AlarmWarnUnAck := FALSE;
   STATUS[597].EXT.AckRequired := FALSE;
   STATUS[597].EXT.Maintanence := FALSE;
   STATUS[597].EXT.Operation := FALSE;
   STATUS[597].EXT.Forced := FALSE;
   STATUS[597].EXT.BIT29 := FALSE;
   STATUS[597].EXT.BIT30 := FALSE;
   STATUS[597].EXT.BIT31 := FALSE;
   STATUS[597].EXT.ModeBit1 := FALSE;
   STATUS[597].EXT.ModeBit2 := FALSE;
   STATUS[597].EXT.ModeBit3 := FALSE;
   STATUS[597].EXT.BIT19 := FALSE;
   STATUS[597].EXT.BIT20 := FALSE;
   STATUS[597].EXT.AlarmSuppressed := FALSE;
   STATUS[597].EXT.AlarmPrsent := FALSE;
   STATUS[597].EXT.AlarmFailUnAck := FALSE;
   STATUS[597].Status := 0;
   STATUS[597].TimeStamp := 16#0000;
   STATUS[598].VALUE := 0.0;
   STATUS[598].TRIGVALUE := 0.0;
   STATUS[598].EXT.AlarmWarnUnAck := FALSE;
   STATUS[598].EXT.AckRequired := FALSE;
   STATUS[598].EXT.Maintanence := FALSE;
   STATUS[598].EXT.Operation := FALSE;
   STATUS[598].EXT.Forced := FALSE;
   STATUS[598].EXT.BIT29 := FALSE;
   STATUS[598].EXT.BIT30 := FALSE;
   STATUS[598].EXT.BIT31 := FALSE;
   STATUS[598].EXT.ModeBit1 := FALSE;
   STATUS[598].EXT.ModeBit2 := FALSE;
   STATUS[598].EXT.ModeBit3 := FALSE;
   STATUS[598].EXT.BIT19 := FALSE;
   STATUS[598].EXT.BIT20 := FALSE;
   STATUS[598].EXT.AlarmSuppressed := FALSE;
   STATUS[598].EXT.AlarmPrsent := FALSE;
   STATUS[598].EXT.AlarmFailUnAck := FALSE;
   STATUS[598].Status := 0;
   STATUS[598].TimeStamp := 16#0000;
   STATUS[599].VALUE := 0.0;
   STATUS[599].TRIGVALUE := 0.0;
   STATUS[599].EXT.AlarmWarnUnAck := FALSE;
   STATUS[599].EXT.AckRequired := FALSE;
   STATUS[599].EXT.Maintanence := FALSE;
   STATUS[599].EXT.Operation := FALSE;
   STATUS[599].EXT.Forced := FALSE;
   STATUS[599].EXT.BIT29 := FALSE;
   STATUS[599].EXT.BIT30 := FALSE;
   STATUS[599].EXT.BIT31 := FALSE;
   STATUS[599].EXT.ModeBit1 := FALSE;
   STATUS[599].EXT.ModeBit2 := FALSE;
   STATUS[599].EXT.ModeBit3 := FALSE;
   STATUS[599].EXT.BIT19 := FALSE;
   STATUS[599].EXT.BIT20 := FALSE;
   STATUS[599].EXT.AlarmSuppressed := FALSE;
   STATUS[599].EXT.AlarmPrsent := FALSE;
   STATUS[599].EXT.AlarmFailUnAck := FALSE;
   STATUS[599].Status := 0;
   STATUS[599].TimeStamp := 16#0000;
   STATUS[600].VALUE := 0.0;
   STATUS[600].TRIGVALUE := 0.0;
   STATUS[600].EXT.AlarmWarnUnAck := FALSE;
   STATUS[600].EXT.AckRequired := FALSE;
   STATUS[600].EXT.Maintanence := FALSE;
   STATUS[600].EXT.Operation := FALSE;
   STATUS[600].EXT.Forced := FALSE;
   STATUS[600].EXT.BIT29 := FALSE;
   STATUS[600].EXT.BIT30 := FALSE;
   STATUS[600].EXT.BIT31 := FALSE;
   STATUS[600].EXT.ModeBit1 := FALSE;
   STATUS[600].EXT.ModeBit2 := FALSE;
   STATUS[600].EXT.ModeBit3 := FALSE;
   STATUS[600].EXT.BIT19 := FALSE;
   STATUS[600].EXT.BIT20 := FALSE;
   STATUS[600].EXT.AlarmSuppressed := FALSE;
   STATUS[600].EXT.AlarmPrsent := FALSE;
   STATUS[600].EXT.AlarmFailUnAck := FALSE;
   STATUS[600].Status := 0;
   STATUS[600].TimeStamp := 16#0000;
   STATUS[601].VALUE := 0.0;
   STATUS[601].TRIGVALUE := 0.0;
   STATUS[601].EXT.AlarmWarnUnAck := FALSE;
   STATUS[601].EXT.AckRequired := FALSE;
   STATUS[601].EXT.Maintanence := FALSE;
   STATUS[601].EXT.Operation := FALSE;
   STATUS[601].EXT.Forced := FALSE;
   STATUS[601].EXT.BIT29 := FALSE;
   STATUS[601].EXT.BIT30 := FALSE;
   STATUS[601].EXT.BIT31 := FALSE;
   STATUS[601].EXT.ModeBit1 := FALSE;
   STATUS[601].EXT.ModeBit2 := FALSE;
   STATUS[601].EXT.ModeBit3 := FALSE;
   STATUS[601].EXT.BIT19 := FALSE;
   STATUS[601].EXT.BIT20 := FALSE;
   STATUS[601].EXT.AlarmSuppressed := FALSE;
   STATUS[601].EXT.AlarmPrsent := FALSE;
   STATUS[601].EXT.AlarmFailUnAck := FALSE;
   STATUS[601].Status := 0;
   STATUS[601].TimeStamp := 16#0000;
   STATUS[602].VALUE := 0.0;
   STATUS[602].TRIGVALUE := 0.0;
   STATUS[602].EXT.AlarmWarnUnAck := FALSE;
   STATUS[602].EXT.AckRequired := FALSE;
   STATUS[602].EXT.Maintanence := FALSE;
   STATUS[602].EXT.Operation := FALSE;
   STATUS[602].EXT.Forced := FALSE;
   STATUS[602].EXT.BIT29 := FALSE;
   STATUS[602].EXT.BIT30 := FALSE;
   STATUS[602].EXT.BIT31 := FALSE;
   STATUS[602].EXT.ModeBit1 := FALSE;
   STATUS[602].EXT.ModeBit2 := FALSE;
   STATUS[602].EXT.ModeBit3 := FALSE;
   STATUS[602].EXT.BIT19 := FALSE;
   STATUS[602].EXT.BIT20 := FALSE;
   STATUS[602].EXT.AlarmSuppressed := FALSE;
   STATUS[602].EXT.AlarmPrsent := FALSE;
   STATUS[602].EXT.AlarmFailUnAck := FALSE;
   STATUS[602].Status := 0;
   STATUS[602].TimeStamp := 16#0000;
   STATUS[603].VALUE := 0.0;
   STATUS[603].TRIGVALUE := 0.0;
   STATUS[603].EXT.AlarmWarnUnAck := FALSE;
   STATUS[603].EXT.AckRequired := FALSE;
   STATUS[603].EXT.Maintanence := FALSE;
   STATUS[603].EXT.Operation := FALSE;
   STATUS[603].EXT.Forced := FALSE;
   STATUS[603].EXT.BIT29 := FALSE;
   STATUS[603].EXT.BIT30 := FALSE;
   STATUS[603].EXT.BIT31 := FALSE;
   STATUS[603].EXT.ModeBit1 := FALSE;
   STATUS[603].EXT.ModeBit2 := FALSE;
   STATUS[603].EXT.ModeBit3 := FALSE;
   STATUS[603].EXT.BIT19 := FALSE;
   STATUS[603].EXT.BIT20 := FALSE;
   STATUS[603].EXT.AlarmSuppressed := FALSE;
   STATUS[603].EXT.AlarmPrsent := FALSE;
   STATUS[603].EXT.AlarmFailUnAck := FALSE;
   STATUS[603].Status := 0;
   STATUS[603].TimeStamp := 16#0000;
   STATUS[604].VALUE := 0.0;
   STATUS[604].TRIGVALUE := 0.0;
   STATUS[604].EXT.AlarmWarnUnAck := FALSE;
   STATUS[604].EXT.AckRequired := FALSE;
   STATUS[604].EXT.Maintanence := FALSE;
   STATUS[604].EXT.Operation := FALSE;
   STATUS[604].EXT.Forced := FALSE;
   STATUS[604].EXT.BIT29 := FALSE;
   STATUS[604].EXT.BIT30 := FALSE;
   STATUS[604].EXT.BIT31 := FALSE;
   STATUS[604].EXT.ModeBit1 := FALSE;
   STATUS[604].EXT.ModeBit2 := FALSE;
   STATUS[604].EXT.ModeBit3 := FALSE;
   STATUS[604].EXT.BIT19 := FALSE;
   STATUS[604].EXT.BIT20 := FALSE;
   STATUS[604].EXT.AlarmSuppressed := FALSE;
   STATUS[604].EXT.AlarmPrsent := FALSE;
   STATUS[604].EXT.AlarmFailUnAck := FALSE;
   STATUS[604].Status := 0;
   STATUS[604].TimeStamp := 16#0000;
   STATUS[605].VALUE := 0.0;
   STATUS[605].TRIGVALUE := 0.0;
   STATUS[605].EXT.AlarmWarnUnAck := FALSE;
   STATUS[605].EXT.AckRequired := FALSE;
   STATUS[605].EXT.Maintanence := FALSE;
   STATUS[605].EXT.Operation := FALSE;
   STATUS[605].EXT.Forced := FALSE;
   STATUS[605].EXT.BIT29 := FALSE;
   STATUS[605].EXT.BIT30 := FALSE;
   STATUS[605].EXT.BIT31 := FALSE;
   STATUS[605].EXT.ModeBit1 := FALSE;
   STATUS[605].EXT.ModeBit2 := FALSE;
   STATUS[605].EXT.ModeBit3 := FALSE;
   STATUS[605].EXT.BIT19 := FALSE;
   STATUS[605].EXT.BIT20 := FALSE;
   STATUS[605].EXT.AlarmSuppressed := FALSE;
   STATUS[605].EXT.AlarmPrsent := FALSE;
   STATUS[605].EXT.AlarmFailUnAck := FALSE;
   STATUS[605].Status := 0;
   STATUS[605].TimeStamp := 16#0000;
   STATUS[606].VALUE := 0.0;
   STATUS[606].TRIGVALUE := 0.0;
   STATUS[606].EXT.AlarmWarnUnAck := FALSE;
   STATUS[606].EXT.AckRequired := FALSE;
   STATUS[606].EXT.Maintanence := FALSE;
   STATUS[606].EXT.Operation := FALSE;
   STATUS[606].EXT.Forced := FALSE;
   STATUS[606].EXT.BIT29 := FALSE;
   STATUS[606].EXT.BIT30 := FALSE;
   STATUS[606].EXT.BIT31 := FALSE;
   STATUS[606].EXT.ModeBit1 := FALSE;
   STATUS[606].EXT.ModeBit2 := FALSE;
   STATUS[606].EXT.ModeBit3 := FALSE;
   STATUS[606].EXT.BIT19 := FALSE;
   STATUS[606].EXT.BIT20 := FALSE;
   STATUS[606].EXT.AlarmSuppressed := FALSE;
   STATUS[606].EXT.AlarmPrsent := FALSE;
   STATUS[606].EXT.AlarmFailUnAck := FALSE;
   STATUS[606].Status := 0;
   STATUS[606].TimeStamp := 16#0000;
   STATUS[607].VALUE := 0.0;
   STATUS[607].TRIGVALUE := 0.0;
   STATUS[607].EXT.AlarmWarnUnAck := FALSE;
   STATUS[607].EXT.AckRequired := FALSE;
   STATUS[607].EXT.Maintanence := FALSE;
   STATUS[607].EXT.Operation := FALSE;
   STATUS[607].EXT.Forced := FALSE;
   STATUS[607].EXT.BIT29 := FALSE;
   STATUS[607].EXT.BIT30 := FALSE;
   STATUS[607].EXT.BIT31 := FALSE;
   STATUS[607].EXT.ModeBit1 := FALSE;
   STATUS[607].EXT.ModeBit2 := FALSE;
   STATUS[607].EXT.ModeBit3 := FALSE;
   STATUS[607].EXT.BIT19 := FALSE;
   STATUS[607].EXT.BIT20 := FALSE;
   STATUS[607].EXT.AlarmSuppressed := FALSE;
   STATUS[607].EXT.AlarmPrsent := FALSE;
   STATUS[607].EXT.AlarmFailUnAck := FALSE;
   STATUS[607].Status := 0;
   STATUS[607].TimeStamp := 16#0000;
   STATUS[608].VALUE := 0.0;
   STATUS[608].TRIGVALUE := 0.0;
   STATUS[608].EXT.AlarmWarnUnAck := FALSE;
   STATUS[608].EXT.AckRequired := FALSE;
   STATUS[608].EXT.Maintanence := FALSE;
   STATUS[608].EXT.Operation := FALSE;
   STATUS[608].EXT.Forced := FALSE;
   STATUS[608].EXT.BIT29 := FALSE;
   STATUS[608].EXT.BIT30 := FALSE;
   STATUS[608].EXT.BIT31 := FALSE;
   STATUS[608].EXT.ModeBit1 := FALSE;
   STATUS[608].EXT.ModeBit2 := FALSE;
   STATUS[608].EXT.ModeBit3 := FALSE;
   STATUS[608].EXT.BIT19 := FALSE;
   STATUS[608].EXT.BIT20 := FALSE;
   STATUS[608].EXT.AlarmSuppressed := FALSE;
   STATUS[608].EXT.AlarmPrsent := FALSE;
   STATUS[608].EXT.AlarmFailUnAck := FALSE;
   STATUS[608].Status := 0;
   STATUS[608].TimeStamp := 16#0000;
   STATUS[609].VALUE := 0.0;
   STATUS[609].TRIGVALUE := 0.0;
   STATUS[609].EXT.AlarmWarnUnAck := FALSE;
   STATUS[609].EXT.AckRequired := FALSE;
   STATUS[609].EXT.Maintanence := FALSE;
   STATUS[609].EXT.Operation := FALSE;
   STATUS[609].EXT.Forced := FALSE;
   STATUS[609].EXT.BIT29 := FALSE;
   STATUS[609].EXT.BIT30 := FALSE;
   STATUS[609].EXT.BIT31 := FALSE;
   STATUS[609].EXT.ModeBit1 := FALSE;
   STATUS[609].EXT.ModeBit2 := FALSE;
   STATUS[609].EXT.ModeBit3 := FALSE;
   STATUS[609].EXT.BIT19 := FALSE;
   STATUS[609].EXT.BIT20 := FALSE;
   STATUS[609].EXT.AlarmSuppressed := FALSE;
   STATUS[609].EXT.AlarmPrsent := FALSE;
   STATUS[609].EXT.AlarmFailUnAck := FALSE;
   STATUS[609].Status := 0;
   STATUS[609].TimeStamp := 16#0000;
   STATUS[610].VALUE := 0.0;
   STATUS[610].TRIGVALUE := 0.0;
   STATUS[610].EXT.AlarmWarnUnAck := FALSE;
   STATUS[610].EXT.AckRequired := FALSE;
   STATUS[610].EXT.Maintanence := FALSE;
   STATUS[610].EXT.Operation := FALSE;
   STATUS[610].EXT.Forced := FALSE;
   STATUS[610].EXT.BIT29 := FALSE;
   STATUS[610].EXT.BIT30 := FALSE;
   STATUS[610].EXT.BIT31 := FALSE;
   STATUS[610].EXT.ModeBit1 := FALSE;
   STATUS[610].EXT.ModeBit2 := FALSE;
   STATUS[610].EXT.ModeBit3 := FALSE;
   STATUS[610].EXT.BIT19 := FALSE;
   STATUS[610].EXT.BIT20 := FALSE;
   STATUS[610].EXT.AlarmSuppressed := FALSE;
   STATUS[610].EXT.AlarmPrsent := FALSE;
   STATUS[610].EXT.AlarmFailUnAck := FALSE;
   STATUS[610].Status := 0;
   STATUS[610].TimeStamp := 16#0000;
   STATUS[611].VALUE := 0.0;
   STATUS[611].TRIGVALUE := 0.0;
   STATUS[611].EXT.AlarmWarnUnAck := FALSE;
   STATUS[611].EXT.AckRequired := FALSE;
   STATUS[611].EXT.Maintanence := FALSE;
   STATUS[611].EXT.Operation := FALSE;
   STATUS[611].EXT.Forced := FALSE;
   STATUS[611].EXT.BIT29 := FALSE;
   STATUS[611].EXT.BIT30 := FALSE;
   STATUS[611].EXT.BIT31 := FALSE;
   STATUS[611].EXT.ModeBit1 := FALSE;
   STATUS[611].EXT.ModeBit2 := FALSE;
   STATUS[611].EXT.ModeBit3 := FALSE;
   STATUS[611].EXT.BIT19 := FALSE;
   STATUS[611].EXT.BIT20 := FALSE;
   STATUS[611].EXT.AlarmSuppressed := FALSE;
   STATUS[611].EXT.AlarmPrsent := FALSE;
   STATUS[611].EXT.AlarmFailUnAck := FALSE;
   STATUS[611].Status := 0;
   STATUS[611].TimeStamp := 16#0000;
   STATUS[612].VALUE := 0.0;
   STATUS[612].TRIGVALUE := 0.0;
   STATUS[612].EXT.AlarmWarnUnAck := FALSE;
   STATUS[612].EXT.AckRequired := FALSE;
   STATUS[612].EXT.Maintanence := FALSE;
   STATUS[612].EXT.Operation := FALSE;
   STATUS[612].EXT.Forced := FALSE;
   STATUS[612].EXT.BIT29 := FALSE;
   STATUS[612].EXT.BIT30 := FALSE;
   STATUS[612].EXT.BIT31 := FALSE;
   STATUS[612].EXT.ModeBit1 := FALSE;
   STATUS[612].EXT.ModeBit2 := FALSE;
   STATUS[612].EXT.ModeBit3 := FALSE;
   STATUS[612].EXT.BIT19 := FALSE;
   STATUS[612].EXT.BIT20 := FALSE;
   STATUS[612].EXT.AlarmSuppressed := FALSE;
   STATUS[612].EXT.AlarmPrsent := FALSE;
   STATUS[612].EXT.AlarmFailUnAck := FALSE;
   STATUS[612].Status := 0;
   STATUS[612].TimeStamp := 16#0000;
   STATUS[613].VALUE := 0.0;
   STATUS[613].TRIGVALUE := 0.0;
   STATUS[613].EXT.AlarmWarnUnAck := FALSE;
   STATUS[613].EXT.AckRequired := FALSE;
   STATUS[613].EXT.Maintanence := FALSE;
   STATUS[613].EXT.Operation := FALSE;
   STATUS[613].EXT.Forced := FALSE;
   STATUS[613].EXT.BIT29 := FALSE;
   STATUS[613].EXT.BIT30 := FALSE;
   STATUS[613].EXT.BIT31 := FALSE;
   STATUS[613].EXT.ModeBit1 := FALSE;
   STATUS[613].EXT.ModeBit2 := FALSE;
   STATUS[613].EXT.ModeBit3 := FALSE;
   STATUS[613].EXT.BIT19 := FALSE;
   STATUS[613].EXT.BIT20 := FALSE;
   STATUS[613].EXT.AlarmSuppressed := FALSE;
   STATUS[613].EXT.AlarmPrsent := FALSE;
   STATUS[613].EXT.AlarmFailUnAck := FALSE;
   STATUS[613].Status := 0;
   STATUS[613].TimeStamp := 16#0000;
   STATUS[614].VALUE := 0.0;
   STATUS[614].TRIGVALUE := 0.0;
   STATUS[614].EXT.AlarmWarnUnAck := FALSE;
   STATUS[614].EXT.AckRequired := FALSE;
   STATUS[614].EXT.Maintanence := FALSE;
   STATUS[614].EXT.Operation := FALSE;
   STATUS[614].EXT.Forced := FALSE;
   STATUS[614].EXT.BIT29 := FALSE;
   STATUS[614].EXT.BIT30 := FALSE;
   STATUS[614].EXT.BIT31 := FALSE;
   STATUS[614].EXT.ModeBit1 := FALSE;
   STATUS[614].EXT.ModeBit2 := FALSE;
   STATUS[614].EXT.ModeBit3 := FALSE;
   STATUS[614].EXT.BIT19 := FALSE;
   STATUS[614].EXT.BIT20 := FALSE;
   STATUS[614].EXT.AlarmSuppressed := FALSE;
   STATUS[614].EXT.AlarmPrsent := FALSE;
   STATUS[614].EXT.AlarmFailUnAck := FALSE;
   STATUS[614].Status := 0;
   STATUS[614].TimeStamp := 16#0000;
   STATUS[615].VALUE := 0.0;
   STATUS[615].TRIGVALUE := 0.0;
   STATUS[615].EXT.AlarmWarnUnAck := FALSE;
   STATUS[615].EXT.AckRequired := FALSE;
   STATUS[615].EXT.Maintanence := FALSE;
   STATUS[615].EXT.Operation := FALSE;
   STATUS[615].EXT.Forced := FALSE;
   STATUS[615].EXT.BIT29 := FALSE;
   STATUS[615].EXT.BIT30 := FALSE;
   STATUS[615].EXT.BIT31 := FALSE;
   STATUS[615].EXT.ModeBit1 := FALSE;
   STATUS[615].EXT.ModeBit2 := FALSE;
   STATUS[615].EXT.ModeBit3 := FALSE;
   STATUS[615].EXT.BIT19 := FALSE;
   STATUS[615].EXT.BIT20 := FALSE;
   STATUS[615].EXT.AlarmSuppressed := FALSE;
   STATUS[615].EXT.AlarmPrsent := FALSE;
   STATUS[615].EXT.AlarmFailUnAck := FALSE;
   STATUS[615].Status := 0;
   STATUS[615].TimeStamp := 16#0000;
   STATUS[616].VALUE := 0.0;
   STATUS[616].TRIGVALUE := 0.0;
   STATUS[616].EXT.AlarmWarnUnAck := FALSE;
   STATUS[616].EXT.AckRequired := FALSE;
   STATUS[616].EXT.Maintanence := FALSE;
   STATUS[616].EXT.Operation := FALSE;
   STATUS[616].EXT.Forced := FALSE;
   STATUS[616].EXT.BIT29 := FALSE;
   STATUS[616].EXT.BIT30 := FALSE;
   STATUS[616].EXT.BIT31 := FALSE;
   STATUS[616].EXT.ModeBit1 := FALSE;
   STATUS[616].EXT.ModeBit2 := FALSE;
   STATUS[616].EXT.ModeBit3 := FALSE;
   STATUS[616].EXT.BIT19 := FALSE;
   STATUS[616].EXT.BIT20 := FALSE;
   STATUS[616].EXT.AlarmSuppressed := FALSE;
   STATUS[616].EXT.AlarmPrsent := FALSE;
   STATUS[616].EXT.AlarmFailUnAck := FALSE;
   STATUS[616].Status := 0;
   STATUS[616].TimeStamp := 16#0000;
   STATUS[617].VALUE := 0.0;
   STATUS[617].TRIGVALUE := 0.0;
   STATUS[617].EXT.AlarmWarnUnAck := FALSE;
   STATUS[617].EXT.AckRequired := FALSE;
   STATUS[617].EXT.Maintanence := FALSE;
   STATUS[617].EXT.Operation := FALSE;
   STATUS[617].EXT.Forced := FALSE;
   STATUS[617].EXT.BIT29 := FALSE;
   STATUS[617].EXT.BIT30 := FALSE;
   STATUS[617].EXT.BIT31 := FALSE;
   STATUS[617].EXT.ModeBit1 := FALSE;
   STATUS[617].EXT.ModeBit2 := FALSE;
   STATUS[617].EXT.ModeBit3 := FALSE;
   STATUS[617].EXT.BIT19 := FALSE;
   STATUS[617].EXT.BIT20 := FALSE;
   STATUS[617].EXT.AlarmSuppressed := FALSE;
   STATUS[617].EXT.AlarmPrsent := FALSE;
   STATUS[617].EXT.AlarmFailUnAck := FALSE;
   STATUS[617].Status := 0;
   STATUS[617].TimeStamp := 16#0000;
   STATUS[618].VALUE := 0.0;
   STATUS[618].TRIGVALUE := 0.0;
   STATUS[618].EXT.AlarmWarnUnAck := FALSE;
   STATUS[618].EXT.AckRequired := FALSE;
   STATUS[618].EXT.Maintanence := FALSE;
   STATUS[618].EXT.Operation := FALSE;
   STATUS[618].EXT.Forced := FALSE;
   STATUS[618].EXT.BIT29 := FALSE;
   STATUS[618].EXT.BIT30 := FALSE;
   STATUS[618].EXT.BIT31 := FALSE;
   STATUS[618].EXT.ModeBit1 := FALSE;
   STATUS[618].EXT.ModeBit2 := FALSE;
   STATUS[618].EXT.ModeBit3 := FALSE;
   STATUS[618].EXT.BIT19 := FALSE;
   STATUS[618].EXT.BIT20 := FALSE;
   STATUS[618].EXT.AlarmSuppressed := FALSE;
   STATUS[618].EXT.AlarmPrsent := FALSE;
   STATUS[618].EXT.AlarmFailUnAck := FALSE;
   STATUS[618].Status := 0;
   STATUS[618].TimeStamp := 16#0000;
   STATUS[619].VALUE := 0.0;
   STATUS[619].TRIGVALUE := 0.0;
   STATUS[619].EXT.AlarmWarnUnAck := FALSE;
   STATUS[619].EXT.AckRequired := FALSE;
   STATUS[619].EXT.Maintanence := FALSE;
   STATUS[619].EXT.Operation := FALSE;
   STATUS[619].EXT.Forced := FALSE;
   STATUS[619].EXT.BIT29 := FALSE;
   STATUS[619].EXT.BIT30 := FALSE;
   STATUS[619].EXT.BIT31 := FALSE;
   STATUS[619].EXT.ModeBit1 := FALSE;
   STATUS[619].EXT.ModeBit2 := FALSE;
   STATUS[619].EXT.ModeBit3 := FALSE;
   STATUS[619].EXT.BIT19 := FALSE;
   STATUS[619].EXT.BIT20 := FALSE;
   STATUS[619].EXT.AlarmSuppressed := FALSE;
   STATUS[619].EXT.AlarmPrsent := FALSE;
   STATUS[619].EXT.AlarmFailUnAck := FALSE;
   STATUS[619].Status := 0;
   STATUS[619].TimeStamp := 16#0000;
   STATUS[620].VALUE := 0.0;
   STATUS[620].TRIGVALUE := 0.0;
   STATUS[620].EXT.AlarmWarnUnAck := FALSE;
   STATUS[620].EXT.AckRequired := FALSE;
   STATUS[620].EXT.Maintanence := FALSE;
   STATUS[620].EXT.Operation := FALSE;
   STATUS[620].EXT.Forced := FALSE;
   STATUS[620].EXT.BIT29 := FALSE;
   STATUS[620].EXT.BIT30 := FALSE;
   STATUS[620].EXT.BIT31 := FALSE;
   STATUS[620].EXT.ModeBit1 := FALSE;
   STATUS[620].EXT.ModeBit2 := FALSE;
   STATUS[620].EXT.ModeBit3 := FALSE;
   STATUS[620].EXT.BIT19 := FALSE;
   STATUS[620].EXT.BIT20 := FALSE;
   STATUS[620].EXT.AlarmSuppressed := FALSE;
   STATUS[620].EXT.AlarmPrsent := FALSE;
   STATUS[620].EXT.AlarmFailUnAck := FALSE;
   STATUS[620].Status := 0;
   STATUS[620].TimeStamp := 16#0000;
   STATUS[621].VALUE := 0.0;
   STATUS[621].TRIGVALUE := 0.0;
   STATUS[621].EXT.AlarmWarnUnAck := FALSE;
   STATUS[621].EXT.AckRequired := FALSE;
   STATUS[621].EXT.Maintanence := FALSE;
   STATUS[621].EXT.Operation := FALSE;
   STATUS[621].EXT.Forced := FALSE;
   STATUS[621].EXT.BIT29 := FALSE;
   STATUS[621].EXT.BIT30 := FALSE;
   STATUS[621].EXT.BIT31 := FALSE;
   STATUS[621].EXT.ModeBit1 := FALSE;
   STATUS[621].EXT.ModeBit2 := FALSE;
   STATUS[621].EXT.ModeBit3 := FALSE;
   STATUS[621].EXT.BIT19 := FALSE;
   STATUS[621].EXT.BIT20 := FALSE;
   STATUS[621].EXT.AlarmSuppressed := FALSE;
   STATUS[621].EXT.AlarmPrsent := FALSE;
   STATUS[621].EXT.AlarmFailUnAck := FALSE;
   STATUS[621].Status := 0;
   STATUS[621].TimeStamp := 16#0000;
   STATUS[622].VALUE := 0.0;
   STATUS[622].TRIGVALUE := 0.0;
   STATUS[622].EXT.AlarmWarnUnAck := FALSE;
   STATUS[622].EXT.AckRequired := FALSE;
   STATUS[622].EXT.Maintanence := FALSE;
   STATUS[622].EXT.Operation := FALSE;
   STATUS[622].EXT.Forced := FALSE;
   STATUS[622].EXT.BIT29 := FALSE;
   STATUS[622].EXT.BIT30 := FALSE;
   STATUS[622].EXT.BIT31 := FALSE;
   STATUS[622].EXT.ModeBit1 := FALSE;
   STATUS[622].EXT.ModeBit2 := FALSE;
   STATUS[622].EXT.ModeBit3 := FALSE;
   STATUS[622].EXT.BIT19 := FALSE;
   STATUS[622].EXT.BIT20 := FALSE;
   STATUS[622].EXT.AlarmSuppressed := FALSE;
   STATUS[622].EXT.AlarmPrsent := FALSE;
   STATUS[622].EXT.AlarmFailUnAck := FALSE;
   STATUS[622].Status := 0;
   STATUS[622].TimeStamp := 16#0000;
   STATUS[623].VALUE := 0.0;
   STATUS[623].TRIGVALUE := 0.0;
   STATUS[623].EXT.AlarmWarnUnAck := FALSE;
   STATUS[623].EXT.AckRequired := FALSE;
   STATUS[623].EXT.Maintanence := FALSE;
   STATUS[623].EXT.Operation := FALSE;
   STATUS[623].EXT.Forced := FALSE;
   STATUS[623].EXT.BIT29 := FALSE;
   STATUS[623].EXT.BIT30 := FALSE;
   STATUS[623].EXT.BIT31 := FALSE;
   STATUS[623].EXT.ModeBit1 := FALSE;
   STATUS[623].EXT.ModeBit2 := FALSE;
   STATUS[623].EXT.ModeBit3 := FALSE;
   STATUS[623].EXT.BIT19 := FALSE;
   STATUS[623].EXT.BIT20 := FALSE;
   STATUS[623].EXT.AlarmSuppressed := FALSE;
   STATUS[623].EXT.AlarmPrsent := FALSE;
   STATUS[623].EXT.AlarmFailUnAck := FALSE;
   STATUS[623].Status := 0;
   STATUS[623].TimeStamp := 16#0000;
   STATUS[624].VALUE := 0.0;
   STATUS[624].TRIGVALUE := 0.0;
   STATUS[624].EXT.AlarmWarnUnAck := FALSE;
   STATUS[624].EXT.AckRequired := FALSE;
   STATUS[624].EXT.Maintanence := FALSE;
   STATUS[624].EXT.Operation := FALSE;
   STATUS[624].EXT.Forced := FALSE;
   STATUS[624].EXT.BIT29 := FALSE;
   STATUS[624].EXT.BIT30 := FALSE;
   STATUS[624].EXT.BIT31 := FALSE;
   STATUS[624].EXT.ModeBit1 := FALSE;
   STATUS[624].EXT.ModeBit2 := FALSE;
   STATUS[624].EXT.ModeBit3 := FALSE;
   STATUS[624].EXT.BIT19 := FALSE;
   STATUS[624].EXT.BIT20 := FALSE;
   STATUS[624].EXT.AlarmSuppressed := FALSE;
   STATUS[624].EXT.AlarmPrsent := FALSE;
   STATUS[624].EXT.AlarmFailUnAck := FALSE;
   STATUS[624].Status := 0;
   STATUS[624].TimeStamp := 16#0000;
   STATUS[625].VALUE := 0.0;
   STATUS[625].TRIGVALUE := 0.0;
   STATUS[625].EXT.AlarmWarnUnAck := FALSE;
   STATUS[625].EXT.AckRequired := FALSE;
   STATUS[625].EXT.Maintanence := FALSE;
   STATUS[625].EXT.Operation := FALSE;
   STATUS[625].EXT.Forced := FALSE;
   STATUS[625].EXT.BIT29 := FALSE;
   STATUS[625].EXT.BIT30 := FALSE;
   STATUS[625].EXT.BIT31 := FALSE;
   STATUS[625].EXT.ModeBit1 := FALSE;
   STATUS[625].EXT.ModeBit2 := FALSE;
   STATUS[625].EXT.ModeBit3 := FALSE;
   STATUS[625].EXT.BIT19 := FALSE;
   STATUS[625].EXT.BIT20 := FALSE;
   STATUS[625].EXT.AlarmSuppressed := FALSE;
   STATUS[625].EXT.AlarmPrsent := FALSE;
   STATUS[625].EXT.AlarmFailUnAck := FALSE;
   STATUS[625].Status := 0;
   STATUS[625].TimeStamp := 16#0000;
   STATUS[626].VALUE := 0.0;
   STATUS[626].TRIGVALUE := 0.0;
   STATUS[626].EXT.AlarmWarnUnAck := FALSE;
   STATUS[626].EXT.AckRequired := FALSE;
   STATUS[626].EXT.Maintanence := FALSE;
   STATUS[626].EXT.Operation := FALSE;
   STATUS[626].EXT.Forced := FALSE;
   STATUS[626].EXT.BIT29 := FALSE;
   STATUS[626].EXT.BIT30 := FALSE;
   STATUS[626].EXT.BIT31 := FALSE;
   STATUS[626].EXT.ModeBit1 := FALSE;
   STATUS[626].EXT.ModeBit2 := FALSE;
   STATUS[626].EXT.ModeBit3 := FALSE;
   STATUS[626].EXT.BIT19 := FALSE;
   STATUS[626].EXT.BIT20 := FALSE;
   STATUS[626].EXT.AlarmSuppressed := FALSE;
   STATUS[626].EXT.AlarmPrsent := FALSE;
   STATUS[626].EXT.AlarmFailUnAck := FALSE;
   STATUS[626].Status := 0;
   STATUS[626].TimeStamp := 16#0000;
   STATUS[627].VALUE := 0.0;
   STATUS[627].TRIGVALUE := 0.0;
   STATUS[627].EXT.AlarmWarnUnAck := FALSE;
   STATUS[627].EXT.AckRequired := FALSE;
   STATUS[627].EXT.Maintanence := FALSE;
   STATUS[627].EXT.Operation := FALSE;
   STATUS[627].EXT.Forced := FALSE;
   STATUS[627].EXT.BIT29 := FALSE;
   STATUS[627].EXT.BIT30 := FALSE;
   STATUS[627].EXT.BIT31 := FALSE;
   STATUS[627].EXT.ModeBit1 := FALSE;
   STATUS[627].EXT.ModeBit2 := FALSE;
   STATUS[627].EXT.ModeBit3 := FALSE;
   STATUS[627].EXT.BIT19 := FALSE;
   STATUS[627].EXT.BIT20 := FALSE;
   STATUS[627].EXT.AlarmSuppressed := FALSE;
   STATUS[627].EXT.AlarmPrsent := FALSE;
   STATUS[627].EXT.AlarmFailUnAck := FALSE;
   STATUS[627].Status := 0;
   STATUS[627].TimeStamp := 16#0000;
   STATUS[628].VALUE := 0.0;
   STATUS[628].TRIGVALUE := 0.0;
   STATUS[628].EXT.AlarmWarnUnAck := FALSE;
   STATUS[628].EXT.AckRequired := FALSE;
   STATUS[628].EXT.Maintanence := FALSE;
   STATUS[628].EXT.Operation := FALSE;
   STATUS[628].EXT.Forced := FALSE;
   STATUS[628].EXT.BIT29 := FALSE;
   STATUS[628].EXT.BIT30 := FALSE;
   STATUS[628].EXT.BIT31 := FALSE;
   STATUS[628].EXT.ModeBit1 := FALSE;
   STATUS[628].EXT.ModeBit2 := FALSE;
   STATUS[628].EXT.ModeBit3 := FALSE;
   STATUS[628].EXT.BIT19 := FALSE;
   STATUS[628].EXT.BIT20 := FALSE;
   STATUS[628].EXT.AlarmSuppressed := FALSE;
   STATUS[628].EXT.AlarmPrsent := FALSE;
   STATUS[628].EXT.AlarmFailUnAck := FALSE;
   STATUS[628].Status := 0;
   STATUS[628].TimeStamp := 16#0000;
   STATUS[629].VALUE := 0.0;
   STATUS[629].TRIGVALUE := 0.0;
   STATUS[629].EXT.AlarmWarnUnAck := FALSE;
   STATUS[629].EXT.AckRequired := FALSE;
   STATUS[629].EXT.Maintanence := FALSE;
   STATUS[629].EXT.Operation := FALSE;
   STATUS[629].EXT.Forced := FALSE;
   STATUS[629].EXT.BIT29 := FALSE;
   STATUS[629].EXT.BIT30 := FALSE;
   STATUS[629].EXT.BIT31 := FALSE;
   STATUS[629].EXT.ModeBit1 := FALSE;
   STATUS[629].EXT.ModeBit2 := FALSE;
   STATUS[629].EXT.ModeBit3 := FALSE;
   STATUS[629].EXT.BIT19 := FALSE;
   STATUS[629].EXT.BIT20 := FALSE;
   STATUS[629].EXT.AlarmSuppressed := FALSE;
   STATUS[629].EXT.AlarmPrsent := FALSE;
   STATUS[629].EXT.AlarmFailUnAck := FALSE;
   STATUS[629].Status := 0;
   STATUS[629].TimeStamp := 16#0000;
   STATUS[630].VALUE := 0.0;
   STATUS[630].TRIGVALUE := 0.0;
   STATUS[630].EXT.AlarmWarnUnAck := FALSE;
   STATUS[630].EXT.AckRequired := FALSE;
   STATUS[630].EXT.Maintanence := FALSE;
   STATUS[630].EXT.Operation := FALSE;
   STATUS[630].EXT.Forced := FALSE;
   STATUS[630].EXT.BIT29 := FALSE;
   STATUS[630].EXT.BIT30 := FALSE;
   STATUS[630].EXT.BIT31 := FALSE;
   STATUS[630].EXT.ModeBit1 := FALSE;
   STATUS[630].EXT.ModeBit2 := FALSE;
   STATUS[630].EXT.ModeBit3 := FALSE;
   STATUS[630].EXT.BIT19 := FALSE;
   STATUS[630].EXT.BIT20 := FALSE;
   STATUS[630].EXT.AlarmSuppressed := FALSE;
   STATUS[630].EXT.AlarmPrsent := FALSE;
   STATUS[630].EXT.AlarmFailUnAck := FALSE;
   STATUS[630].Status := 0;
   STATUS[630].TimeStamp := 16#0000;
   STATUS[631].VALUE := 0.0;
   STATUS[631].TRIGVALUE := 0.0;
   STATUS[631].EXT.AlarmWarnUnAck := FALSE;
   STATUS[631].EXT.AckRequired := FALSE;
   STATUS[631].EXT.Maintanence := FALSE;
   STATUS[631].EXT.Operation := FALSE;
   STATUS[631].EXT.Forced := FALSE;
   STATUS[631].EXT.BIT29 := FALSE;
   STATUS[631].EXT.BIT30 := FALSE;
   STATUS[631].EXT.BIT31 := FALSE;
   STATUS[631].EXT.ModeBit1 := FALSE;
   STATUS[631].EXT.ModeBit2 := FALSE;
   STATUS[631].EXT.ModeBit3 := FALSE;
   STATUS[631].EXT.BIT19 := FALSE;
   STATUS[631].EXT.BIT20 := FALSE;
   STATUS[631].EXT.AlarmSuppressed := FALSE;
   STATUS[631].EXT.AlarmPrsent := FALSE;
   STATUS[631].EXT.AlarmFailUnAck := FALSE;
   STATUS[631].Status := 0;
   STATUS[631].TimeStamp := 16#0000;
   STATUS[632].VALUE := 0.0;
   STATUS[632].TRIGVALUE := 0.0;
   STATUS[632].EXT.AlarmWarnUnAck := FALSE;
   STATUS[632].EXT.AckRequired := FALSE;
   STATUS[632].EXT.Maintanence := FALSE;
   STATUS[632].EXT.Operation := FALSE;
   STATUS[632].EXT.Forced := FALSE;
   STATUS[632].EXT.BIT29 := FALSE;
   STATUS[632].EXT.BIT30 := FALSE;
   STATUS[632].EXT.BIT31 := FALSE;
   STATUS[632].EXT.ModeBit1 := FALSE;
   STATUS[632].EXT.ModeBit2 := FALSE;
   STATUS[632].EXT.ModeBit3 := FALSE;
   STATUS[632].EXT.BIT19 := FALSE;
   STATUS[632].EXT.BIT20 := FALSE;
   STATUS[632].EXT.AlarmSuppressed := FALSE;
   STATUS[632].EXT.AlarmPrsent := FALSE;
   STATUS[632].EXT.AlarmFailUnAck := FALSE;
   STATUS[632].Status := 0;
   STATUS[632].TimeStamp := 16#0000;
   STATUS[633].VALUE := 0.0;
   STATUS[633].TRIGVALUE := 0.0;
   STATUS[633].EXT.AlarmWarnUnAck := FALSE;
   STATUS[633].EXT.AckRequired := FALSE;
   STATUS[633].EXT.Maintanence := FALSE;
   STATUS[633].EXT.Operation := FALSE;
   STATUS[633].EXT.Forced := FALSE;
   STATUS[633].EXT.BIT29 := FALSE;
   STATUS[633].EXT.BIT30 := FALSE;
   STATUS[633].EXT.BIT31 := FALSE;
   STATUS[633].EXT.ModeBit1 := FALSE;
   STATUS[633].EXT.ModeBit2 := FALSE;
   STATUS[633].EXT.ModeBit3 := FALSE;
   STATUS[633].EXT.BIT19 := FALSE;
   STATUS[633].EXT.BIT20 := FALSE;
   STATUS[633].EXT.AlarmSuppressed := FALSE;
   STATUS[633].EXT.AlarmPrsent := FALSE;
   STATUS[633].EXT.AlarmFailUnAck := FALSE;
   STATUS[633].Status := 0;
   STATUS[633].TimeStamp := 16#0000;
   STATUS[634].VALUE := 0.0;
   STATUS[634].TRIGVALUE := 0.0;
   STATUS[634].EXT.AlarmWarnUnAck := FALSE;
   STATUS[634].EXT.AckRequired := FALSE;
   STATUS[634].EXT.Maintanence := FALSE;
   STATUS[634].EXT.Operation := FALSE;
   STATUS[634].EXT.Forced := FALSE;
   STATUS[634].EXT.BIT29 := FALSE;
   STATUS[634].EXT.BIT30 := FALSE;
   STATUS[634].EXT.BIT31 := FALSE;
   STATUS[634].EXT.ModeBit1 := FALSE;
   STATUS[634].EXT.ModeBit2 := FALSE;
   STATUS[634].EXT.ModeBit3 := FALSE;
   STATUS[634].EXT.BIT19 := FALSE;
   STATUS[634].EXT.BIT20 := FALSE;
   STATUS[634].EXT.AlarmSuppressed := FALSE;
   STATUS[634].EXT.AlarmPrsent := FALSE;
   STATUS[634].EXT.AlarmFailUnAck := FALSE;
   STATUS[634].Status := 0;
   STATUS[634].TimeStamp := 16#0000;
   STATUS[635].VALUE := 0.0;
   STATUS[635].TRIGVALUE := 0.0;
   STATUS[635].EXT.AlarmWarnUnAck := FALSE;
   STATUS[635].EXT.AckRequired := FALSE;
   STATUS[635].EXT.Maintanence := FALSE;
   STATUS[635].EXT.Operation := FALSE;
   STATUS[635].EXT.Forced := FALSE;
   STATUS[635].EXT.BIT29 := FALSE;
   STATUS[635].EXT.BIT30 := FALSE;
   STATUS[635].EXT.BIT31 := FALSE;
   STATUS[635].EXT.ModeBit1 := FALSE;
   STATUS[635].EXT.ModeBit2 := FALSE;
   STATUS[635].EXT.ModeBit3 := FALSE;
   STATUS[635].EXT.BIT19 := FALSE;
   STATUS[635].EXT.BIT20 := FALSE;
   STATUS[635].EXT.AlarmSuppressed := FALSE;
   STATUS[635].EXT.AlarmPrsent := FALSE;
   STATUS[635].EXT.AlarmFailUnAck := FALSE;
   STATUS[635].Status := 0;
   STATUS[635].TimeStamp := 16#0000;
   STATUS[636].VALUE := 0.0;
   STATUS[636].TRIGVALUE := 0.0;
   STATUS[636].EXT.AlarmWarnUnAck := FALSE;
   STATUS[636].EXT.AckRequired := FALSE;
   STATUS[636].EXT.Maintanence := FALSE;
   STATUS[636].EXT.Operation := FALSE;
   STATUS[636].EXT.Forced := FALSE;
   STATUS[636].EXT.BIT29 := FALSE;
   STATUS[636].EXT.BIT30 := FALSE;
   STATUS[636].EXT.BIT31 := FALSE;
   STATUS[636].EXT.ModeBit1 := FALSE;
   STATUS[636].EXT.ModeBit2 := FALSE;
   STATUS[636].EXT.ModeBit3 := FALSE;
   STATUS[636].EXT.BIT19 := FALSE;
   STATUS[636].EXT.BIT20 := FALSE;
   STATUS[636].EXT.AlarmSuppressed := FALSE;
   STATUS[636].EXT.AlarmPrsent := FALSE;
   STATUS[636].EXT.AlarmFailUnAck := FALSE;
   STATUS[636].Status := 0;
   STATUS[636].TimeStamp := 16#0000;
   STATUS[637].VALUE := 0.0;
   STATUS[637].TRIGVALUE := 0.0;
   STATUS[637].EXT.AlarmWarnUnAck := FALSE;
   STATUS[637].EXT.AckRequired := FALSE;
   STATUS[637].EXT.Maintanence := FALSE;
   STATUS[637].EXT.Operation := FALSE;
   STATUS[637].EXT.Forced := FALSE;
   STATUS[637].EXT.BIT29 := FALSE;
   STATUS[637].EXT.BIT30 := FALSE;
   STATUS[637].EXT.BIT31 := FALSE;
   STATUS[637].EXT.ModeBit1 := FALSE;
   STATUS[637].EXT.ModeBit2 := FALSE;
   STATUS[637].EXT.ModeBit3 := FALSE;
   STATUS[637].EXT.BIT19 := FALSE;
   STATUS[637].EXT.BIT20 := FALSE;
   STATUS[637].EXT.AlarmSuppressed := FALSE;
   STATUS[637].EXT.AlarmPrsent := FALSE;
   STATUS[637].EXT.AlarmFailUnAck := FALSE;
   STATUS[637].Status := 0;
   STATUS[637].TimeStamp := 16#0000;
   STATUS[638].VALUE := 0.0;
   STATUS[638].TRIGVALUE := 0.0;
   STATUS[638].EXT.AlarmWarnUnAck := FALSE;
   STATUS[638].EXT.AckRequired := FALSE;
   STATUS[638].EXT.Maintanence := FALSE;
   STATUS[638].EXT.Operation := FALSE;
   STATUS[638].EXT.Forced := FALSE;
   STATUS[638].EXT.BIT29 := FALSE;
   STATUS[638].EXT.BIT30 := FALSE;
   STATUS[638].EXT.BIT31 := FALSE;
   STATUS[638].EXT.ModeBit1 := FALSE;
   STATUS[638].EXT.ModeBit2 := FALSE;
   STATUS[638].EXT.ModeBit3 := FALSE;
   STATUS[638].EXT.BIT19 := FALSE;
   STATUS[638].EXT.BIT20 := FALSE;
   STATUS[638].EXT.AlarmSuppressed := FALSE;
   STATUS[638].EXT.AlarmPrsent := FALSE;
   STATUS[638].EXT.AlarmFailUnAck := FALSE;
   STATUS[638].Status := 0;
   STATUS[638].TimeStamp := 16#0000;
   STATUS[639].VALUE := 0.0;
   STATUS[639].TRIGVALUE := 0.0;
   STATUS[639].EXT.AlarmWarnUnAck := FALSE;
   STATUS[639].EXT.AckRequired := FALSE;
   STATUS[639].EXT.Maintanence := FALSE;
   STATUS[639].EXT.Operation := FALSE;
   STATUS[639].EXT.Forced := FALSE;
   STATUS[639].EXT.BIT29 := FALSE;
   STATUS[639].EXT.BIT30 := FALSE;
   STATUS[639].EXT.BIT31 := FALSE;
   STATUS[639].EXT.ModeBit1 := FALSE;
   STATUS[639].EXT.ModeBit2 := FALSE;
   STATUS[639].EXT.ModeBit3 := FALSE;
   STATUS[639].EXT.BIT19 := FALSE;
   STATUS[639].EXT.BIT20 := FALSE;
   STATUS[639].EXT.AlarmSuppressed := FALSE;
   STATUS[639].EXT.AlarmPrsent := FALSE;
   STATUS[639].EXT.AlarmFailUnAck := FALSE;
   STATUS[639].Status := 0;
   STATUS[639].TimeStamp := 16#0000;
   STATUS[640].VALUE := 0.0;
   STATUS[640].TRIGVALUE := 0.0;
   STATUS[640].EXT.AlarmWarnUnAck := FALSE;
   STATUS[640].EXT.AckRequired := FALSE;
   STATUS[640].EXT.Maintanence := FALSE;
   STATUS[640].EXT.Operation := FALSE;
   STATUS[640].EXT.Forced := FALSE;
   STATUS[640].EXT.BIT29 := FALSE;
   STATUS[640].EXT.BIT30 := FALSE;
   STATUS[640].EXT.BIT31 := FALSE;
   STATUS[640].EXT.ModeBit1 := FALSE;
   STATUS[640].EXT.ModeBit2 := FALSE;
   STATUS[640].EXT.ModeBit3 := FALSE;
   STATUS[640].EXT.BIT19 := FALSE;
   STATUS[640].EXT.BIT20 := FALSE;
   STATUS[640].EXT.AlarmSuppressed := FALSE;
